LIN {X -0.024,Y -228.688,Z 374.177,A 0.000,B 0.000,C 90.000,E1 31.848} C_DIS
LIN {X 0.017,Y -219.940,Z 374.156,A 0.000,B 0.000,C 90.000,E1 28.025} C_DIS
LIN {X -0.020,Y -212.162,Z 374.134,A 0.000,B 0.000,C 90.000,E1 24.155} C_DIS
LIN {X 0.098,Y -206.724,Z 374.117,A 0.000,B 0.000,C 90.000,E1 20.972} C_DIS
LIN {X -0.105,Y -200.813,Z 374.095,A 0.000,B 0.000,C 90.000,E1 17.040} C_DIS
LIN {X 0.032,Y -196.763,Z 374.077,A 0.000,B 0.000,C 90.000,E1 13.772} C_DIS
LIN {X -0.062,Y -192.666,Z 374.054,A 0.000,B 0.000,C 90.000,E1 9.726} C_DIS
LIN {X -0.090,Y -189.777,Z 374.031,A 0.000,B 0.000,C 90.000,E1 5.625} C_DIS
LIN {X 0.062,Y -187.714,Z 373.993,A 0.000,B 0.000,C 90.000,E1 358.682} C_DIS
LIN {X 0.002,Y -189.474,Z 373.942,A 0.000,B 0.000,C 90.000,E1 349.577} C_DIS
LIN {X -0.013,Y -192.481,Z 373.915,A 0.000,B 0.000,C 90.000,E1 344.629} C_DIS
LIN {X -0.083,Y -196.181,Z 373.892,A 0.000,B 0.000,C 90.000,E1 340.550} C_DIS
LIN {X -0.079,Y -200.966,Z 373.869,A 0.000,B 0.000,C 90.000,E1 336.485} C_DIS
LIN {X -0.043,Y -205.596,Z 373.851,A 0.000,B 0.000,C 90.000,E1 333.256} C_DIS
LIN {X -0.055,Y -212.277,Z 373.829,A 0.000,B 0.000,C 90.000,E1 329.282} C_DIS
LIN {X 0.024,Y -219.465,Z 373.807,A 0.000,B 0.000,C 90.000,E1 325.341} C_DIS
LIN {X -0.061,Y -225.849,Z 373.790,A 0.000,B 0.000,C 90.000,E1 322.271} C_DIS
LIN {X 0.005,Y -234.579,Z 373.769,A 0.000,B 0.000,C 90.000,E1 318.447} C_DIS
LIN {X 0.024,Y -243.663,Z 373.750,A 0.000,B 0.000,C 90.000,E1 315.081} C_DIS
LIN {X -0.040,Y -252.669,Z 373.734,A 0.000,B 0.000,C 90.000,E1 312.162} C_DIS
LIN {X -0.020,Y -262.716,Z 373.718,A 0.000,B 0.000,C 90.000,E1 309.277} C_DIS
LIN {X 0.045,Y -274.656,Z 373.701,A 0.000,B 0.000,C 90.000,E1 306.091} C_DIS
LIN {X -0.160,Y -285.719,Z 373.685,A 0.000,B 0.000,C 90.000,E1 303.372} C_DIS
LIN {X -0.156,Y -299.626,Z 373.668,A 0.000,B 0.000,C 90.000,E1 300.335} C_DIS
LIN {X 0.072,Y -315.196,Z 373.652,A 0.000,B 0.000,C 90.000,E1 297.334} C_DIS
LIN {X 0.056,Y -326.808,Z 373.641,A 0.000,B 0.000,C 90.000,E1 295.412} C_DIS
LIN {X 0.118,Y -339.498,Z 373.631,A 0.000,B 0.000,C 90.000,E1 293.515} C_DIS
LIN {X -0.141,Y -355.051,Z 373.619,A 0.000,B 0.000,C 90.000,E1 291.408} C_DIS
LIN {X 0.226,Y -373.453,Z 373.606,A 0.000,B 0.000,C 90.000,E1 288.960} C_DIS
LIN {X 0.071,Y -398.842,Z 373.590,A 0.000,B 0.000,C 90.000,E1 286.150} C_DIS
LIN {X -0.135,Y -416.958,Z 373.579,A 0.000,B 0.000,C 90.000,E1 284.300} C_DIS
LIN {X -0.034,Y -427.204,Z 373.574,A 0.000,B 0.000,C 90.000,E1 283.244} C_DIS
LIN {X 0.012,Y -437.142,Z 373.568,A 0.000,B 0.000,C 90.000,E1 282.187} C_DIS
LIN {X -0.235,Y -444.156,Z 373.563,A 0.000,B 0.000,C 90.000,E1 281.422} C_DIS
LIN {X -0.195,Y -452.664,Z 373.557,A 0.000,B 0.000,C 90.000,E1 280.366} C_DIS
LIN {X -0.136,Y -460.420,Z 373.552,A 0.000,B 0.000,C 90.000,E1 279.321} C_DIS
LIN {X 0.014,Y -467.426,Z 373.546,A 0.000,B 0.000,C 90.000,E1 278.276} C_DIS
LIN {X 0.186,Y -473.852,Z 373.540,A 0.000,B 0.000,C 90.000,E1 277.239} C_DIS
LIN {X -0.034,Y -479.682,Z 373.535,A 0.000,B 0.000,C 90.000,E1 276.258} C_DIS
LIN {X -0.063,Y -483.421,Z 373.531,A 0.000,B 0.000,C 90.000,E1 275.511} C_DIS
LIN {X 0.114,Y -485.523,Z 373.528,A 0.000,B 0.000,C 90.000,E1 274.992} C_DIS
LIN {X -0.181,Y -487.261,Z 373.525,A 0.000,B 0.000,C 90.000,E1 274.531} C_DIS
LIN {X 0.011,Y -488.621,Z 373.522,A 0.000,B 0.000,C 90.000,E1 274.012} C_DIS
LIN {X 0.181,Y -489.646,Z 373.520,A 0.000,B 0.000,C 90.000,E1 273.498} C_DIS
LIN {X -0.100,Y -490.325,Z 373.517,A 0.000,B 0.000,C 90.000,E1 273.037} C_DIS
LIN {X 0.089,Y -490.720,Z 373.514,A 0.000,B 0.000,C 90.000,E1 272.522} C_DIS
LIN {X -0.206,Y -490.827,Z 373.511,A 0.000,B 0.000,C 90.000,E1 272.064} C_DIS
LIN {X 0.007,Y -490.615,Z 373.509,A 0.000,B 0.000,C 90.000,E1 271.547} C_DIS
LIN {X 0.205,Y -490.110,Z 373.506,A 0.000,B 0.000,C 90.000,E1 271.031} C_DIS
LIN {X -0.086,Y -489.189,Z 373.503,A 0.000,B 0.000,C 90.000,E1 270.573} C_DIS
LIN {X 0.110,Y -487.799,Z 373.500,A 0.000,B 0.000,C 90.000,E1 270.057} C_DIS
LIN {X -0.186,Y -485.830,Z 373.498,A 0.000,B 0.000,C 90.000,E1 269.599} C_DIS
LIN {X 0.148,Y -484.659,Z 373.496,A 0.000,B 0.000,C 90.000,E1 269.312} C_DIS
LIN {X -0.165,Y -481.666,Z 373.494,A 0.000,B 0.000,C 90.000,E1 268.854} C_DIS
LIN {X -0.013,Y -477.763,Z 373.491,A 0.000,B 0.000,C 90.000,E1 268.339} C_DIS
LIN {X -0.165,Y -475.427,Z 373.489,A 0.000,B 0.000,C 90.000,E1 268.108} C_DIS
LIN {X -0.044,Y -469.718,Z 373.487,A 0.000,B 0.000,C 90.000,E1 267.593} C_DIS
LIN {X 0.107,Y -463.235,Z 373.484,A 0.000,B 0.000,C 90.000,E1 267.135} C_DIS
LIN {X 0.020,Y -459.955,Z 373.483,A 0.000,B 0.000,C 90.000,E1 266.963} C_DIS
LIN {X 0.177,Y -452.875,Z 373.481,A 0.000,B 0.000,C 90.000,E1 266.617} C_DIS
LIN {X -0.068,Y -445.562,Z 373.480,A 0.000,B 0.000,C 90.000,E1 266.388} C_DIS
LIN {X 0.108,Y -437.885,Z 373.479,A 0.000,B 0.000,C 90.000,E1 266.159} C_DIS
LIN {X -0.210,Y -429.466,Z 373.478,A 0.000,B 0.000,C 90.000,E1 266.045} C_DIS
LIN {X -0.134,Y -418.655,Z 373.477,A 0.000,B 0.000,C 90.000,E1 265.927} C_DIS
LIN {X 0.128,Y -414.372,Z 373.477,A 0.000,B 0.000,C 90.000,E1 265.869} C_DIS
LIN {X 0.023,Y -180.915,Z 373.477,A 0.000,B 0.000,C 90.000,E1 265.869} C_DIS
LIN {X 0.051,Y -180.822,Z 373.471,A 0.000,B 0.000,C 90.000,E1 264.837} C_DIS
LIN {X -0.054,Y -178.854,Z 373.442,A 0.000,B 0.000,C 90.000,E1 259.634} C_DIS
LIN {X 0.017,Y -175.897,Z 373.414,A 0.000,B 0.000,C 90.000,E1 254.519} C_DIS
LIN {X -0.044,Y -174.574,Z 373.405,A 0.000,B 0.000,C 90.000,E1 252.834} C_DIS
LIN {X -0.008,Y -171.557,Z 373.381,A 0.000,B 0.000,C 90.000,E1 248.539} C_DIS
LIN {X 0.048,Y -167.781,Z 373.357,A 0.000,B 0.000,C 90.000,E1 244.204} C_DIS
LIN {X -0.011,Y -166.494,Z 373.347,A 0.000,B 0.000,C 90.000,E1 242.487} C_DIS
LIN {X -0.015,Y -163.204,Z 373.328,A 0.000,B 0.000,C 90.000,E1 238.997} C_DIS
LIN {X 0.039,Y -161.168,Z 373.313,A 0.000,B 0.000,C 90.000,E1 236.342} C_DIS
LIN {X 0.074,Y -157.183,Z 373.289,A 0.000,B 0.000,C 90.000,E1 231.904} C_DIS
LIN {X -0.003,Y -155.912,Z 373.279,A 0.000,B 0.000,C 90.000,E1 230.150} C_DIS
LIN {X 0.053,Y -152.163,Z 373.254,A 0.000,B 0.000,C 90.000,E1 225.648} C_DIS
LIN {X 0.073,Y -150.412,Z 373.239,A 0.000,B 0.000,C 90.000,E1 222.933} C_DIS
LIN {X 0.004,Y -147.141,Z 373.213,A 0.000,B 0.000,C 90.000,E1 218.418} C_DIS
LIN {X 0.002,Y -145.700,Z 373.198,A 0.000,B 0.000,C 90.000,E1 215.678} C_DIS
LIN {X 0.009,Y -143.083,Z 373.173,A 0.000,B 0.000,C 90.000,E1 211.082} C_DIS
LIN {X 0.014,Y -141.701,Z 373.152,A 0.000,B 0.000,C 90.000,E1 207.385} C_DIS
LIN {X -0.063,Y -139.467,Z 373.116,A 0.000,B 0.000,C 90.000,E1 200.918} C_DIS
LIN {X -0.010,Y -139.200,Z 373.106,A 0.000,B 0.000,C 90.000,E1 199.033} C_DIS
LIN {X 0.054,Y -138.327,Z 373.054,A 0.000,B 0.000,C 90.000,E1 189.670} C_DIS
LIN {X 0.059,Y -139.445,Z 373.007,A 0.000,B 0.000,C 90.000,E1 181.260} C_DIS
LIN {X 0.000,Y -140.983,Z 372.976,A 0.000,B 0.000,C 90.000,E1 175.698} C_DIS
LIN {X -0.051,Y -142.739,Z 372.955,A 0.000,B 0.000,C 90.000,E1 172.008} C_DIS
LIN {X 0.047,Y -145.131,Z 372.930,A 0.000,B 0.000,C 90.000,E1 167.353} C_DIS
LIN {X 0.042,Y -147.754,Z 372.909,A 0.000,B 0.000,C 90.000,E1 163.685} C_DIS
LIN {X -0.020,Y -150.424,Z 372.889,A 0.000,B 0.000,C 90.000,E1 160.061} C_DIS
LIN {X -0.005,Y -153.865,Z 372.869,A 0.000,B 0.000,C 90.000,E1 156.433} C_DIS
LIN {X -0.088,Y -157.276,Z 372.849,A 0.000,B 0.000,C 90.000,E1 152.871} C_DIS
LIN {X -0.011,Y -161.454,Z 372.829,A 0.000,B 0.000,C 90.000,E1 149.282} C_DIS
LIN {X -0.004,Y -165.655,Z 372.810,A 0.000,B 0.000,C 90.000,E1 145.754} C_DIS
LIN {X -0.022,Y -170.590,Z 372.790,A 0.000,B 0.000,C 90.000,E1 142.271} C_DIS
LIN {X 0.017,Y -175.468,Z 372.771,A 0.000,B 0.000,C 90.000,E1 138.809} C_DIS
LIN {X 0.000,Y -181.090,Z 372.752,A 0.000,B 0.000,C 90.000,E1 135.405} C_DIS
LIN {X -0.010,Y -186.531,Z 372.734,A 0.000,B 0.000,C 90.000,E1 132.043} C_DIS
LIN {X -0.069,Y -191.149,Z 372.720,A 0.000,B 0.000,C 90.000,E1 129.564} C_DIS
LIN {X 0.009,Y -196.950,Z 372.701,A 0.000,B 0.000,C 90.000,E1 126.251} C_DIS
LIN {X -0.085,Y -199.016,Z 372.696,A 0.000,B 0.000,C 90.000,E1 125.231} C_DIS
LIN {X 0.067,Y -298.976,Z 372.696,A 0.000,B 0.000,C 90.000,E1 125.185} C_DIS
LIN {X -0.082,Y -300.521,Z 372.695,A 0.000,B 0.000,C 90.000,E1 125.185} C_DIS
LIN {X -0.007,Y -305.764,Z 372.694,A 0.000,B 0.000,C 90.000,E1 124.898} C_DIS
LIN {X 0.070,Y -308.564,Z 372.692,A 0.000,B 0.000,C 90.000,E1 124.612} C_DIS
LIN {X 0.009,Y -312.276,Z 372.689,A 0.000,B 0.000,C 90.000,E1 124.072} C_DIS
LIN {X -0.208,Y -313.814,Z 372.688,A 0.000,B 0.000,C 90.000,E1 123.785} C_DIS
LIN {X 0.077,Y -320.564,Z 372.677,A 0.000,B 0.000,C 90.000,E1 121.799} C_DIS
LIN {X 0.040,Y -331.559,Z 372.661,A 0.000,B 0.000,C 90.000,E1 118.949} C_DIS
LIN {X -0.002,Y -343.956,Z 372.645,A 0.000,B 0.000,C 90.000,E1 116.155} C_DIS
LIN {X 0.123,Y -356.250,Z 372.632,A 0.000,B 0.000,C 90.000,E1 113.695} C_DIS
LIN {X -0.057,Y -369.833,Z 372.618,A 0.000,B 0.000,C 90.000,E1 111.334} C_DIS
LIN {X 0.186,Y -384.804,Z 372.605,A 0.000,B 0.000,C 90.000,E1 108.960} C_DIS
LIN {X 0.205,Y -401.275,Z 372.593,A 0.000,B 0.000,C 90.000,E1 106.677} C_DIS
LIN {X 0.020,Y -419.367,Z 372.580,A 0.000,B 0.000,C 90.000,E1 104.481} C_DIS
LIN {X -0.114,Y -439.036,Z 372.569,A 0.000,B 0.000,C 90.000,E1 102.355} C_DIS
LIN {X -0.027,Y -459.428,Z 372.558,A 0.000,B 0.000,C 90.000,E1 100.366} C_DIS
LIN {X -0.068,Y -482.997,Z 372.546,A 0.000,B 0.000,C 90.000,E1 98.341} C_DIS
LIN {X -0.008,Y -490.879,Z 372.543,A 0.000,B 0.000,C 90.000,E1 97.701} C_DIS
LIN {X 0.157,Y -492.885,Z 372.542,A 0.000,B 0.000,C 90.000,E1 97.473} C_DIS
LIN {X 0.059,Y -494.681,Z 372.540,A 0.000,B 0.000,C 90.000,E1 97.239} C_DIS
LIN {X -0.042,Y -496.029,Z 372.539,A 0.000,B 0.000,C 90.000,E1 97.004} C_DIS
LIN {X 0.210,Y -497.710,Z 372.536,A 0.000,B 0.000,C 90.000,E1 96.486} C_DIS
LIN {X -0.078,Y -498.302,Z 372.533,A 0.000,B 0.000,C 90.000,E1 96.030} C_DIS
LIN {X 0.194,Y -497.899,Z 372.531,A 0.000,B 0.000,C 90.000,E1 95.511} C_DIS
LIN {X -0.027,Y -496.437,Z 372.528,A 0.000,B 0.000,C 90.000,E1 95.049} C_DIS
LIN {X -0.159,Y -495.229,Z 372.527,A 0.000,B 0.000,C 90.000,E1 94.821} C_DIS
LIN {X -0.035,Y -490.066,Z 372.523,A 0.000,B 0.000,C 90.000,E1 94.073} C_DIS
LIN {X -0.087,Y -482.358,Z 372.517,A 0.000,B 0.000,C 90.000,E1 93.094} C_DIS
LIN {X -0.201,Y -460.635,Z 372.502,A 0.000,B 0.000,C 90.000,E1 90.344} C_DIS
LIN {X 0.204,Y -442.378,Z 372.487,A 0.000,B 0.000,C 90.000,E1 87.707} C_DIS
LIN {X 0.098,Y -420.907,Z 372.468,A 0.000,B 0.000,C 90.000,E1 84.261} C_DIS
LIN {X -0.157,Y -407.216,Z 372.455,A 0.000,B 0.000,C 90.000,E1 81.837} C_DIS
LIN {X 0.072,Y -395.395,Z 372.442,A 0.000,B 0.000,C 90.000,E1 79.577} C_DIS
LIN {X 0.110,Y -385.202,Z 372.431,A 0.000,B 0.000,C 90.000,E1 77.589} C_DIS
LIN {X 0.118,Y -372.056,Z 372.417,A 0.000,B 0.000,C 90.000,E1 74.991} C_DIS
LIN {X -0.087,Y -360.570,Z 372.404,A 0.000,B 0.000,C 90.000,E1 72.670} C_DIS
LIN {X 0.067,Y -350.621,Z 372.392,A 0.000,B 0.000,C 90.000,E1 70.550} C_DIS
LIN {X 0.131,Y -338.104,Z 372.377,A 0.000,B 0.000,C 90.000,E1 67.794} C_DIS
LIN {X -0.137,Y -323.705,Z 372.358,A 0.000,B 0.000,C 90.000,E1 64.409} C_DIS
LIN {X 0.065,Y -311.675,Z 372.340,A 0.000,B 0.000,C 90.000,E1 61.179} C_DIS
LIN {X 0.081,Y -300.462,Z 372.322,A 0.000,B 0.000,C 90.000,E1 57.916} C_DIS
LIN {X 0.017,Y -290.095,Z 372.303,A 0.000,B 0.000,C 90.000,E1 54.609} C_DIS
LIN {X 0.042,Y -282.469,Z 372.288,A 0.000,B 0.000,C 90.000,E1 51.904} C_DIS
LIN {X -0.003,Y -275.091,Z 372.273,A 0.000,B 0.000,C 90.000,E1 49.175} C_DIS
LIN {X 0.095,Y -267.499,Z 372.258,A 0.000,B 0.000,C 90.000,E1 46.377} C_DIS
LIN {X -0.002,Y -259.878,Z 372.242,A 0.000,B 0.000,C 90.000,E1 43.581} C_DIS
LIN {X 0.029,Y -254.052,Z 372.230,A 0.000,B 0.000,C 90.000,E1 41.434} C_DIS
LIN {X 0.020,Y -246.068,Z 372.214,A 0.000,B 0.000,C 90.000,E1 38.543} C_DIS
LIN {X 0.051,Y -238.246,Z 372.198,A 0.000,B 0.000,C 90.000,E1 35.598} C_DIS
LIN {X 0.000,Y -230.723,Z 372.181,A 0.000,B 0.000,C 90.000,E1 32.625} C_DIS
LIN {X 0.021,Y -223.507,Z 372.164,A 0.000,B 0.000,C 90.000,E1 29.589} C_DIS
LIN {X 0.111,Y -216.892,Z 372.147,A 0.000,B 0.000,C 90.000,E1 26.488} C_DIS
LIN {X 0.043,Y -210.870,Z 372.130,A 0.000,B 0.000,C 90.000,E1 23.387} C_DIS
LIN {X -0.030,Y -205.581,Z 372.112,A 0.000,B 0.000,C 90.000,E1 20.248} C_DIS
LIN {X -0.069,Y -199.789,Z 372.090,A 0.000,B 0.000,C 90.000,E1 16.260} C_DIS
LIN {X -0.007,Y -195.947,Z 372.072,A 0.000,B 0.000,C 90.000,E1 13.008} C_DIS
LIN {X 0.027,Y -192.016,Z 372.050,A 0.000,B 0.000,C 90.000,E1 8.916} C_DIS
LIN {X 0.091,Y -188.997,Z 372.022,A 0.000,B 0.000,C 90.000,E1 3.955} C_DIS
LIN {X -0.067,Y -188.058,Z 371.965,A 0.000,B 0.000,C 90.000,E1 353.742} C_DIS
LIN {X -0.066,Y -190.713,Z 371.928,A 0.000,B 0.000,C 90.000,E1 347.117} C_DIS
LIN {X -0.070,Y -194.489,Z 371.901,A 0.000,B 0.000,C 90.000,E1 342.181} C_DIS
LIN {X -0.076,Y -198.867,Z 371.878,A 0.000,B 0.000,C 90.000,E1 338.103} C_DIS
LIN {X 0.006,Y -203.091,Z 371.860,A 0.000,B 0.000,C 90.000,E1 334.845} C_DIS
LIN {X 0.007,Y -209.442,Z 371.838,A 0.000,B 0.000,C 90.000,E1 330.845} C_DIS
LIN {X -0.039,Y -216.434,Z 371.816,A 0.000,B 0.000,C 90.000,E1 326.914} C_DIS
LIN {X 0.031,Y -222.445,Z 371.799,A 0.000,B 0.000,C 90.000,E1 323.783} C_DIS
LIN {X -0.015,Y -229.178,Z 371.782,A 0.000,B 0.000,C 90.000,E1 320.723} C_DIS
LIN {X 0.018,Y -237.396,Z 371.763,A 0.000,B 0.000,C 90.000,E1 317.310} C_DIS
LIN {X 0.115,Y -246.852,Z 371.744,A 0.000,B 0.000,C 90.000,E1 313.947} C_DIS
LIN {X 0.111,Y -253.839,Z 371.732,A 0.000,B 0.000,C 90.000,E1 311.757} C_DIS
LIN {X -0.006,Y -263.914,Z 371.716,A 0.000,B 0.000,C 90.000,E1 308.910} C_DIS
LIN {X 0.007,Y -274.572,Z 371.701,A 0.000,B 0.000,C 90.000,E1 306.091} C_DIS
LIN {X 0.194,Y -285.683,Z 371.685,A 0.000,B 0.000,C 90.000,E1 303.293} C_DIS
LIN {X 0.059,Y -299.634,Z 371.668,A 0.000,B 0.000,C 90.000,E1 300.285} C_DIS
LIN {X 0.027,Y -315.307,Z 371.652,A 0.000,B 0.000,C 90.000,E1 297.334} C_DIS
LIN {X 0.074,Y -324.949,Z 371.643,A 0.000,B 0.000,C 90.000,E1 295.720} C_DIS
LIN {X 0.076,Y -339.679,Z 371.631,A 0.000,B 0.000,C 90.000,E1 293.515} C_DIS
LIN {X -0.181,Y -355.254,Z 371.619,A 0.000,B 0.000,C 90.000,E1 291.408} C_DIS
LIN {X 0.098,Y -371.302,Z 371.607,A 0.000,B 0.000,C 90.000,E1 289.268} C_DIS
LIN {X -0.168,Y -386.166,Z 371.598,A 0.000,B 0.000,C 90.000,E1 287.583} C_DIS
LIN {X 0.020,Y -404.328,Z 371.587,A 0.000,B 0.000,C 90.000,E1 285.607} C_DIS
LIN {X -0.243,Y -422.490,Z 371.576,A 0.000,B 0.000,C 90.000,E1 283.772} C_DIS
LIN {X 0.041,Y -432.438,Z 371.571,A 0.000,B 0.000,C 90.000,E1 282.703} C_DIS
LIN {X -0.206,Y -439.634,Z 371.566,A 0.000,B 0.000,C 90.000,E1 281.951} C_DIS
LIN {X 0.063,Y -446.350,Z 371.562,A 0.000,B 0.000,C 90.000,E1 281.130} C_DIS
LIN {X 0.134,Y -454.649,Z 371.556,A 0.000,B 0.000,C 90.000,E1 280.074} C_DIS
LIN {X 0.221,Y -462.124,Z 371.550,A 0.000,B 0.000,C 90.000,E1 279.029} C_DIS
LIN {X -0.134,Y -469.004,Z 371.545,A 0.000,B 0.000,C 90.000,E1 278.049} C_DIS
LIN {X 0.119,Y -475.230,Z 371.539,A 0.000,B 0.000,C 90.000,E1 277.004} C_DIS
LIN {X 0.051,Y -479.565,Z 371.535,A 0.000,B 0.000,C 90.000,E1 276.258} C_DIS
LIN {X 0.020,Y -483.335,Z 371.531,A 0.000,B 0.000,C 90.000,E1 275.511} C_DIS
LIN {X 0.198,Y -485.450,Z 371.528,A 0.000,B 0.000,C 90.000,E1 274.992} C_DIS
LIN {X -0.098,Y -487.170,Z 371.525,A 0.000,B 0.000,C 90.000,E1 274.531} C_DIS
LIN {X 0.094,Y -488.544,Z 371.522,A 0.000,B 0.000,C 90.000,E1 274.012} C_DIS
LIN {X -0.225,Y -489.539,Z 371.520,A 0.000,B 0.000,C 90.000,E1 273.555} C_DIS
LIN {X -0.018,Y -490.211,Z 371.517,A 0.000,B 0.000,C 90.000,E1 273.037} C_DIS
LIN {X 0.171,Y -490.608,Z 371.514,A 0.000,B 0.000,C 90.000,E1 272.522} C_DIS
LIN {X -0.125,Y -490.705,Z 371.511,A 0.000,B 0.000,C 90.000,E1 272.064} C_DIS
LIN {X 0.088,Y -490.499,Z 371.509,A 0.000,B 0.000,C 90.000,E1 271.547} C_DIS
LIN {X -0.204,Y -489.981,Z 371.506,A 0.000,B 0.000,C 90.000,E1 271.088} C_DIS
LIN {X -0.006,Y -489.061,Z 371.503,A 0.000,B 0.000,C 90.000,E1 270.573} C_DIS
LIN {X 0.188,Y -487.719,Z 371.500,A 0.000,B 0.000,C 90.000,E1 270.057} C_DIS
LIN {X -0.109,Y -485.816,Z 371.498,A 0.000,B 0.000,C 90.000,E1 269.599} C_DIS
LIN {X 0.072,Y -483.222,Z 371.495,A 0.000,B 0.000,C 90.000,E1 269.083} C_DIS
LIN {X -0.089,Y -481.681,Z 371.494,A 0.000,B 0.000,C 90.000,E1 268.854} C_DIS
LIN {X 0.062,Y -477.860,Z 371.491,A 0.000,B 0.000,C 90.000,E1 268.339} C_DIS
LIN {X -0.090,Y -475.546,Z 371.489,A 0.000,B 0.000,C 90.000,E1 268.108} C_DIS
LIN {X 0.208,Y -472.879,Z 371.488,A 0.000,B 0.000,C 90.000,E1 267.822} C_DIS
LIN {X 0.098,Y -466.953,Z 371.485,A 0.000,B 0.000,C 90.000,E1 267.364} C_DIS
LIN {X 0.107,Y -460.313,Z 371.483,A 0.000,B 0.000,C 90.000,E1 266.963} C_DIS
LIN {X -0.206,Y -453.387,Z 371.481,A 0.000,B 0.000,C 90.000,E1 266.674} C_DIS
LIN {X -0.054,Y -445.982,Z 371.480,A 0.000,B 0.000,C 90.000,E1 266.388} C_DIS
LIN {X 0.104,Y -438.346,Z 371.479,A 0.000,B 0.000,C 90.000,E1 266.159} C_DIS
LIN {X -0.225,Y -429.948,Z 371.478,A 0.000,B 0.000,C 90.000,E1 266.045} C_DIS
LIN {X -0.156,Y -419.101,Z 371.477,A 0.000,B 0.000,C 90.000,E1 265.927} C_DIS
LIN {X 0.106,Y -415.628,Z 371.477,A 0.000,B 0.000,C 90.000,E1 265.869} C_DIS
LIN {X 0.012,Y -180.915,Z 371.477,A 0.000,B 0.000,C 90.000,E1 265.869} C_DIS
LIN {X 0.040,Y -180.821,Z 371.471,A 0.000,B 0.000,C 90.000,E1 264.837} C_DIS
LIN {X -0.065,Y -178.852,Z 371.442,A 0.000,B 0.000,C 90.000,E1 259.634} C_DIS
LIN {X 0.007,Y -175.896,Z 371.414,A 0.000,B 0.000,C 90.000,E1 254.519} C_DIS
LIN {X -0.055,Y -174.571,Z 371.405,A 0.000,B 0.000,C 90.000,E1 252.834} C_DIS
LIN {X -0.019,Y -171.554,Z 371.381,A 0.000,B 0.000,C 90.000,E1 248.539} C_DIS
LIN {X 0.037,Y -167.778,Z 371.357,A 0.000,B 0.000,C 90.000,E1 244.204} C_DIS
LIN {X -0.021,Y -166.490,Z 371.347,A 0.000,B 0.000,C 90.000,E1 242.487} C_DIS
LIN {X -0.026,Y -163.200,Z 371.328,A 0.000,B 0.000,C 90.000,E1 238.997} C_DIS
LIN {X 0.028,Y -161.164,Z 371.313,A 0.000,B 0.000,C 90.000,E1 236.342} C_DIS
LIN {X 0.064,Y -157.180,Z 371.288,A 0.000,B 0.000,C 90.000,E1 231.904} C_DIS
LIN {X -0.014,Y -155.910,Z 371.279,A 0.000,B 0.000,C 90.000,E1 230.150} C_DIS
LIN {X 0.043,Y -152.161,Z 371.254,A 0.000,B 0.000,C 90.000,E1 225.648} C_DIS
LIN {X 0.063,Y -150.410,Z 371.239,A 0.000,B 0.000,C 90.000,E1 222.933} C_DIS
LIN {X 0.086,Y -147.139,Z 371.213,A 0.000,B 0.000,C 90.000,E1 218.382} C_DIS
LIN {X -0.008,Y -145.698,Z 371.198,A 0.000,B 0.000,C 90.000,E1 215.678} C_DIS
LIN {X 0.000,Y -143.082,Z 371.173,A 0.000,B 0.000,C 90.000,E1 211.082} C_DIS
LIN {X 0.004,Y -141.699,Z 371.152,A 0.000,B 0.000,C 90.000,E1 207.385} C_DIS
LIN {X -0.073,Y -139.466,Z 371.116,A 0.000,B 0.000,C 90.000,E1 200.918} C_DIS
LIN {X -0.019,Y -139.199,Z 371.106,A 0.000,B 0.000,C 90.000,E1 199.033} C_DIS
LIN {X 0.045,Y -138.327,Z 371.054,A 0.000,B 0.000,C 90.000,E1 189.670} C_DIS
LIN {X 0.050,Y -139.446,Z 371.007,A 0.000,B 0.000,C 90.000,E1 181.260} C_DIS
LIN {X -0.010,Y -140.985,Z 370.976,A 0.000,B 0.000,C 90.000,E1 175.698} C_DIS
LIN {X -0.060,Y -142.740,Z 370.955,A 0.000,B 0.000,C 90.000,E1 172.008} C_DIS
LIN {X 0.038,Y -145.133,Z 370.930,A 0.000,B 0.000,C 90.000,E1 167.353} C_DIS
LIN {X 0.031,Y -147.756,Z 370.909,A 0.000,B 0.000,C 90.000,E1 163.685} C_DIS
LIN {X -0.029,Y -150.426,Z 370.889,A 0.000,B 0.000,C 90.000,E1 160.061} C_DIS
LIN {X -0.015,Y -153.869,Z 370.869,A 0.000,B 0.000,C 90.000,E1 156.433} C_DIS
LIN {X 0.042,Y -157.280,Z 370.849,A 0.000,B 0.000,C 90.000,E1 152.820} C_DIS
LIN {X -0.021,Y -161.459,Z 370.829,A 0.000,B 0.000,C 90.000,E1 149.282} C_DIS
LIN {X -0.015,Y -165.660,Z 370.810,A 0.000,B 0.000,C 90.000,E1 145.754} C_DIS
LIN {X -0.033,Y -170.596,Z 370.790,A 0.000,B 0.000,C 90.000,E1 142.271} C_DIS
LIN {X 0.005,Y -175.472,Z 370.771,A 0.000,B 0.000,C 90.000,E1 138.809} C_DIS
LIN {X -0.011,Y -181.095,Z 370.752,A 0.000,B 0.000,C 90.000,E1 135.405} C_DIS
LIN {X -0.022,Y -186.538,Z 370.734,A 0.000,B 0.000,C 90.000,E1 132.043} C_DIS
LIN {X -0.081,Y -191.154,Z 370.720,A 0.000,B 0.000,C 90.000,E1 129.564} C_DIS
LIN {X -0.003,Y -196.957,Z 370.701,A 0.000,B 0.000,C 90.000,E1 126.251} C_DIS
LIN {X 0.000,Y -199.129,Z 370.695,A 0.000,B 0.000,C 90.000,E1 125.152} C_DIS
LIN {X -0.036,Y -298.758,Z 370.695,A 0.000,B 0.000,C 90.000,E1 125.152} C_DIS
LIN {X -0.018,Y -301.092,Z 370.695,A 0.000,B 0.000,C 90.000,E1 125.105} C_DIS
LIN {X -0.022,Y -305.657,Z 370.694,A 0.000,B 0.000,C 90.000,E1 124.865} C_DIS
LIN {X 0.052,Y -308.254,Z 370.692,A 0.000,B 0.000,C 90.000,E1 124.612} C_DIS
LIN {X -0.151,Y -312.031,Z 370.689,A 0.000,B 0.000,C 90.000,E1 124.119} C_DIS
LIN {X -0.109,Y -313.659,Z 370.688,A 0.000,B 0.000,C 90.000,E1 123.785} C_DIS
LIN {X 0.166,Y -316.023,Z 370.684,A 0.000,B 0.000,C 90.000,E1 123.086} C_DIS
LIN {X -0.116,Y -326.417,Z 370.668,A 0.000,B 0.000,C 90.000,E1 120.256} C_DIS
LIN {X 0.146,Y -338.167,Z 370.652,A 0.000,B 0.000,C 90.000,E1 117.385} C_DIS
LIN {X -0.018,Y -351.389,Z 370.637,A 0.000,B 0.000,C 90.000,E1 114.643} C_DIS
LIN {X 0.159,Y -364.468,Z 370.624,A 0.000,B 0.000,C 90.000,E1 112.206} C_DIS
LIN {X -0.080,Y -378.897,Z 370.610,A 0.000,B 0.000,C 90.000,E1 109.885} C_DIS
LIN {X -0.089,Y -394.782,Z 370.598,A 0.000,B 0.000,C 90.000,E1 107.583} C_DIS
LIN {X 0.065,Y -412.240,Z 370.585,A 0.000,B 0.000,C 90.000,E1 105.315} C_DIS
LIN {X 0.155,Y -431.393,Z 370.573,A 0.000,B 0.000,C 90.000,E1 103.119} C_DIS
LIN {X 0.169,Y -451.570,Z 370.562,A 0.000,B 0.000,C 90.000,E1 101.074} C_DIS
LIN {X 0.114,Y -472.289,Z 370.551,A 0.000,B 0.000,C 90.000,E1 99.208} C_DIS
LIN {X 0.082,Y -490.755,Z 370.543,A 0.000,B 0.000,C 90.000,E1 97.701} C_DIS
LIN {X -0.243,Y -492.842,Z 370.542,A 0.000,B 0.000,C 90.000,E1 97.530} C_DIS
LIN {X 0.180,Y -494.676,Z 370.540,A 0.000,B 0.000,C 90.000,E1 97.239} C_DIS
LIN {X 0.113,Y -496.060,Z 370.539,A 0.000,B 0.000,C 90.000,E1 97.004} C_DIS
LIN {X -0.130,Y -497.831,Z 370.536,A 0.000,B 0.000,C 90.000,E1 96.543} C_DIS
LIN {X 0.077,Y -498.496,Z 370.534,A 0.000,B 0.000,C 90.000,E1 96.030} C_DIS
LIN {X -0.146,Y -498.165,Z 370.531,A 0.000,B 0.000,C 90.000,E1 95.568} C_DIS
LIN {X 0.129,Y -496.785,Z 370.528,A 0.000,B 0.000,C 90.000,E1 95.049} C_DIS
LIN {X -0.003,Y -495.629,Z 370.527,A 0.000,B 0.000,C 90.000,E1 94.821} C_DIS
LIN {X -0.232,Y -492.321,Z 370.524,A 0.000,B 0.000,C 90.000,E1 94.359} C_DIS
LIN {X 0.199,Y -484.814,Z 370.519,A 0.000,B 0.000,C 90.000,E1 93.326} C_DIS
LIN {X 0.184,Y -472.799,Z 370.510,A 0.000,B 0.000,C 90.000,E1 91.835} C_DIS
LIN {X 0.004,Y -449.877,Z 370.493,A 0.000,B 0.000,C 90.000,E1 88.797} C_DIS
LIN {X 0.141,Y -427.642,Z 370.474,A 0.000,B 0.000,C 90.000,E1 85.355} C_DIS
LIN {X -0.086,Y -409.071,Z 370.456,A 0.000,B 0.000,C 90.000,E1 82.129} C_DIS
LIN {X -0.131,Y -395.773,Z 370.442,A 0.000,B 0.000,C 90.000,E1 79.634} C_DIS
LIN {X -0.037,Y -384.102,Z 370.430,A 0.000,B 0.000,C 90.000,E1 77.353} C_DIS
LIN {X -0.049,Y -372.424,Z 370.417,A 0.000,B 0.000,C 90.000,E1 75.046} C_DIS
LIN {X 0.109,Y -360.933,Z 370.404,A 0.000,B 0.000,C 90.000,E1 72.670} C_DIS
LIN {X -0.066,Y -350.960,Z 370.392,A 0.000,B 0.000,C 90.000,E1 70.604} C_DIS
LIN {X 0.016,Y -338.382,Z 370.377,A 0.000,B 0.000,C 90.000,E1 67.847} C_DIS
LIN {X 0.063,Y -323.950,Z 370.358,A 0.000,B 0.000,C 90.000,E1 64.409} C_DIS
LIN {X -0.074,Y -313.094,Z 370.342,A 0.000,B 0.000,C 90.000,E1 61.563} C_DIS
LIN {X -0.134,Y -300.706,Z 370.322,A 0.000,B 0.000,C 90.000,E1 57.995} C_DIS
LIN {X 0.044,Y -290.326,Z 370.304,A 0.000,B 0.000,C 90.000,E1 54.642} C_DIS
LIN {X 0.014,Y -282.689,Z 370.289,A 0.000,B 0.000,C 90.000,E1 51.949} C_DIS
LIN {X -0.027,Y -277.135,Z 370.277,A 0.000,B 0.000,C 90.000,E1 49.908} C_DIS
LIN {X -0.029,Y -271.493,Z 370.266,A 0.000,B 0.000,C 90.000,E1 47.838} C_DIS
LIN {X 0.046,Y -265.811,Z 370.254,A 0.000,B 0.000,C 90.000,E1 45.729} C_DIS
LIN {X -0.090,Y -258.174,Z 370.238,A 0.000,B 0.000,C 90.000,E1 42.933} C_DIS
LIN {X -0.071,Y -252.294,Z 370.226,A 0.000,B 0.000,C 90.000,E1 40.782} C_DIS
LIN {X -0.114,Y -244.356,Z 370.210,A 0.000,B 0.000,C 90.000,E1 37.890} C_DIS
LIN {X 0.070,Y -236.592,Z 370.194,A 0.000,B 0.000,C 90.000,E1 34.898} C_DIS
LIN {X -0.024,Y -229.103,Z 370.177,A 0.000,B 0.000,C 90.000,E1 31.926} C_DIS
LIN {X 0.031,Y -221.996,Z 370.160,A 0.000,B 0.000,C 90.000,E1 28.871} C_DIS
LIN {X -0.047,Y -213.969,Z 370.139,A 0.000,B 0.000,C 90.000,E1 25.027} C_DIS
LIN {X -0.076,Y -208.297,Z 370.122,A 0.000,B 0.000,C 90.000,E1 21.897} C_DIS
LIN {X -0.089,Y -203.318,Z 370.104,A 0.000,B 0.000,C 90.000,E1 18.725} C_DIS
LIN {X 0.028,Y -198.843,Z 370.086,A 0.000,B 0.000,C 90.000,E1 15.481} C_DIS
LIN {X 0.036,Y -194.348,Z 370.064,A 0.000,B 0.000,C 90.000,E1 11.422} C_DIS
LIN {X -0.049,Y -190.846,Z 370.041,A 0.000,B 0.000,C 90.000,E1 7.352} C_DIS
LIN {X 0.035,Y -188.140,Z 370.009,A 0.000,B 0.000,C 90.000,E1 1.547} C_DIS
LIN {X 0.032,Y -189.398,Z 369.942,A 0.000,B 0.000,C 90.000,E1 349.567} C_DIS
LIN {X -0.021,Y -192.341,Z 369.915,A 0.000,B 0.000,C 90.000,E1 344.629} C_DIS
LIN {X -0.095,Y -196.034,Z 369.892,A 0.000,B 0.000,C 90.000,E1 340.550} C_DIS
LIN {X -0.097,Y -200.811,Z 369.869,A 0.000,B 0.000,C 90.000,E1 336.485} C_DIS
LIN {X -0.065,Y -205.431,Z 369.851,A 0.000,B 0.000,C 90.000,E1 333.256} C_DIS
LIN {X 0.024,Y -212.092,Z 369.829,A 0.000,B 0.000,C 90.000,E1 329.253} C_DIS
LIN {X -0.011,Y -219.262,Z 369.807,A 0.000,B 0.000,C 90.000,E1 325.341} C_DIS
LIN {X -0.102,Y -225.682,Z 369.790,A 0.000,B 0.000,C 90.000,E1 322.271} C_DIS
LIN {X -0.043,Y -234.424,Z 369.769,A 0.000,B 0.000,C 90.000,E1 318.447} C_DIS
LIN {X -0.031,Y -243.523,Z 369.750,A 0.000,B 0.000,C 90.000,E1 315.081} C_DIS
LIN {X 0.070,Y -252.537,Z 369.734,A 0.000,B 0.000,C 90.000,E1 312.123} C_DIS
LIN {X -0.086,Y -262.544,Z 369.718,A 0.000,B 0.000,C 90.000,E1 309.277} C_DIS
LIN {X -0.029,Y -274.491,Z 369.700,A 0.000,B 0.000,C 90.000,E1 306.091} C_DIS
LIN {X 0.040,Y -284.184,Z 369.687,A 0.000,B 0.000,C 90.000,E1 303.658} C_DIS
LIN {X 0.018,Y -299.654,Z 369.668,A 0.000,B 0.000,C 90.000,E1 300.285} C_DIS
LIN {X 0.083,Y -313.592,Z 369.654,A 0.000,B 0.000,C 90.000,E1 297.641} C_DIS
LIN {X -0.048,Y -323.116,Z 369.645,A 0.000,B 0.000,C 90.000,E1 296.052} C_DIS
LIN {X 0.057,Y -337.672,Z 369.632,A 0.000,B 0.000,C 90.000,E1 293.823} C_DIS
LIN {X 0.077,Y -353.244,Z 369.620,A 0.000,B 0.000,C 90.000,E1 291.663} C_DIS
LIN {X 0.064,Y -371.557,Z 369.607,A 0.000,B 0.000,C 90.000,E1 289.268} C_DIS
LIN {X 0.041,Y -388.930,Z 369.596,A 0.000,B 0.000,C 90.000,E1 287.275} C_DIS
LIN {X -0.084,Y -406.919,Z 369.585,A 0.000,B 0.000,C 90.000,E1 285.371} C_DIS
LIN {X -0.062,Y -422.426,Z 369.576,A 0.000,B 0.000,C 90.000,E1 283.772} C_DIS
LIN {X -0.209,Y -430.022,Z 369.572,A 0.000,B 0.000,C 90.000,E1 283.008} C_DIS
LIN {X 0.014,Y -437.375,Z 369.568,A 0.000,B 0.000,C 90.000,E1 282.187} C_DIS
LIN {X -0.232,Y -444.322,Z 369.563,A 0.000,B 0.000,C 90.000,E1 281.422} C_DIS
LIN {X -0.189,Y -452.716,Z 369.557,A 0.000,B 0.000,C 90.000,E1 280.366} C_DIS
LIN {X 0.051,Y -458.528,Z 369.553,A 0.000,B 0.000,C 90.000,E1 279.557} C_DIS
LIN {X 0.186,Y -465.681,Z 369.547,A 0.000,B 0.000,C 90.000,E1 278.511} C_DIS
LIN {X -0.126,Y -472.185,Z 369.542,A 0.000,B 0.000,C 90.000,E1 277.530} C_DIS
LIN {X 0.164,Y -478.144,Z 369.536,A 0.000,B 0.000,C 90.000,E1 276.486} C_DIS
LIN {X 0.124,Y -482.137,Z 369.532,A 0.000,B 0.000,C 90.000,E1 275.739} C_DIS
LIN {X -0.191,Y -484.418,Z 369.529,A 0.000,B 0.000,C 90.000,E1 275.277} C_DIS
LIN {X -0.179,Y -487.133,Z 369.525,A 0.000,B 0.000,C 90.000,E1 274.531} C_DIS
LIN {X 0.012,Y -488.472,Z 369.522,A 0.000,B 0.000,C 90.000,E1 274.012} C_DIS
LIN {X 0.182,Y -489.462,Z 369.520,A 0.000,B 0.000,C 90.000,E1 273.498} C_DIS
LIN {X -0.099,Y -490.090,Z 369.517,A 0.000,B 0.000,C 90.000,E1 273.037} C_DIS
LIN {X 0.088,Y -490.468,Z 369.514,A 0.000,B 0.000,C 90.000,E1 272.522} C_DIS
LIN {X -0.208,Y -490.560,Z 369.511,A 0.000,B 0.000,C 90.000,E1 272.064} C_DIS
LIN {X 0.003,Y -490.349,Z 369.509,A 0.000,B 0.000,C 90.000,E1 271.547} C_DIS
LIN {X 0.200,Y -489.798,Z 369.506,A 0.000,B 0.000,C 90.000,E1 271.031} C_DIS
LIN {X -0.093,Y -488.890,Z 369.503,A 0.000,B 0.000,C 90.000,E1 270.573} C_DIS
LIN {X 0.101,Y -487.539,Z 369.500,A 0.000,B 0.000,C 90.000,E1 270.057} C_DIS
LIN {X -0.196,Y -485.624,Z 369.498,A 0.000,B 0.000,C 90.000,E1 269.599} C_DIS
LIN {X -0.016,Y -483.072,Z 369.495,A 0.000,B 0.000,C 90.000,E1 269.083} C_DIS
LIN {X 0.143,Y -479.768,Z 369.492,A 0.000,B 0.000,C 90.000,E1 268.568} C_DIS
LIN {X -0.026,Y -477.751,Z 369.491,A 0.000,B 0.000,C 90.000,E1 268.339} C_DIS
LIN {X -0.178,Y -475.453,Z 369.489,A 0.000,B 0.000,C 90.000,E1 268.108} C_DIS
LIN {X -0.057,Y -469.868,Z 369.487,A 0.000,B 0.000,C 90.000,E1 267.593} C_DIS
LIN {X 0.014,Y -463.325,Z 369.484,A 0.000,B 0.000,C 90.000,E1 267.135} C_DIS
LIN {X -0.154,Y -456.402,Z 369.482,A 0.000,B 0.000,C 90.000,E1 266.788} C_DIS
LIN {X 0.194,Y -448.969,Z 369.480,A 0.000,B 0.000,C 90.000,E1 266.445} C_DIS
LIN {X 0.171,Y -441.525,Z 369.479,A 0.000,B 0.000,C 90.000,E1 266.216} C_DIS
LIN {X 0.098,Y -433.241,Z 369.478,A 0.000,B 0.000,C 90.000,E1 266.045} C_DIS
LIN {X 0.035,Y -423.586,Z 369.477,A 0.000,B 0.000,C 90.000,E1 265.927} C_DIS
LIN {X 0.000,Y -412.395,Z 369.477,A 0.000,B 0.000,C 90.000,E1 265.869} C_DIS
LIN {X -0.033,Y -180.915,Z 369.477,A 0.000,B 0.000,C 90.000,E1 265.869} C_DIS
LIN {X -0.003,Y -180.817,Z 369.471,A 0.000,B 0.000,C 90.000,E1 264.837} C_DIS
LIN {X 0.068,Y -178.846,Z 369.442,A 0.000,B 0.000,C 90.000,E1 259.577} C_DIS
LIN {X -0.037,Y -175.889,Z 369.414,A 0.000,B 0.000,C 90.000,E1 254.519} C_DIS
LIN {X 0.070,Y -174.559,Z 369.404,A 0.000,B 0.000,C 90.000,E1 252.779} C_DIS
LIN {X -0.061,Y -171.543,Z 369.381,A 0.000,B 0.000,C 90.000,E1 248.539} C_DIS
LIN {X -0.005,Y -167.768,Z 369.357,A 0.000,B 0.000,C 90.000,E1 244.204} C_DIS
LIN {X -0.064,Y -166.476,Z 369.347,A 0.000,B 0.000,C 90.000,E1 242.487} C_DIS
LIN {X -0.067,Y -163.189,Z 369.328,A 0.000,B 0.000,C 90.000,E1 238.997} C_DIS
LIN {X -0.012,Y -161.150,Z 369.313,A 0.000,B 0.000,C 90.000,E1 236.342} C_DIS
LIN {X 0.024,Y -157.169,Z 369.288,A 0.000,B 0.000,C 90.000,E1 231.904} C_DIS
LIN {X -0.054,Y -155.900,Z 369.279,A 0.000,B 0.000,C 90.000,E1 230.150} C_DIS
LIN {X 0.004,Y -152.149,Z 369.254,A 0.000,B 0.000,C 90.000,E1 225.648} C_DIS
LIN {X 0.023,Y -150.399,Z 369.239,A 0.000,B 0.000,C 90.000,E1 222.933} C_DIS
LIN {X 0.047,Y -147.130,Z 369.213,A 0.000,B 0.000,C 90.000,E1 218.382} C_DIS
LIN {X -0.046,Y -145.692,Z 369.198,A 0.000,B 0.000,C 90.000,E1 215.678} C_DIS
LIN {X 0.036,Y -143.074,Z 369.173,A 0.000,B 0.000,C 90.000,E1 211.052} C_DIS
LIN {X -0.033,Y -141.694,Z 369.152,A 0.000,B 0.000,C 90.000,E1 207.385} C_DIS
LIN {X 0.021,Y -139.463,Z 369.116,A 0.000,B 0.000,C 90.000,E1 200.865} C_DIS
LIN {X -0.056,Y -139.197,Z 369.106,A 0.000,B 0.000,C 90.000,E1 199.033} C_DIS
LIN {X 0.007,Y -138.325,Z 369.054,A 0.000,B 0.000,C 90.000,E1 189.670} C_DIS
LIN {X 0.013,Y -139.449,Z 369.007,A 0.000,B 0.000,C 90.000,E1 181.260} C_DIS
LIN {X -0.048,Y -140.991,Z 368.976,A 0.000,B 0.000,C 90.000,E1 175.698} C_DIS
LIN {X 0.043,Y -142.746,Z 368.955,A 0.000,B 0.000,C 90.000,E1 171.951} C_DIS
LIN {X 0.000,Y -145.143,Z 368.930,A 0.000,B 0.000,C 90.000,E1 167.353} C_DIS
LIN {X -0.007,Y -147.765,Z 368.909,A 0.000,B 0.000,C 90.000,E1 163.685} C_DIS
LIN {X -0.068,Y -150.439,Z 368.889,A 0.000,B 0.000,C 90.000,E1 160.061} C_DIS
LIN {X 0.008,Y -153.885,Z 368.869,A 0.000,B 0.000,C 90.000,E1 156.410} C_DIS
LIN {X 0.002,Y -157.295,Z 368.849,A 0.000,B 0.000,C 90.000,E1 152.820} C_DIS
LIN {X 0.020,Y -161.478,Z 368.829,A 0.000,B 0.000,C 90.000,E1 149.253} C_DIS
LIN {X 0.037,Y -165.677,Z 368.810,A 0.000,B 0.000,C 90.000,E1 145.722} C_DIS
LIN {X -0.076,Y -170.618,Z 368.790,A 0.000,B 0.000,C 90.000,E1 142.271} C_DIS
LIN {X 0.078,Y -175.494,Z 368.771,A 0.000,B 0.000,C 90.000,E1 138.771} C_DIS
LIN {X -0.056,Y -181.115,Z 368.752,A 0.000,B 0.000,C 90.000,E1 135.405} C_DIS
LIN {X 0.072,Y -186.563,Z 368.733,A 0.000,B 0.000,C 90.000,E1 132.000} C_DIS
LIN {X 0.022,Y -191.176,Z 368.720,A 0.000,B 0.000,C 90.000,E1 129.519} C_DIS
LIN {X 0.067,Y -196.982,Z 368.701,A 0.000,B 0.000,C 90.000,E1 126.217} C_DIS
LIN {X -0.028,Y -199.240,Z 368.695,A 0.000,B 0.000,C 90.000,E1 125.105} C_DIS
LIN {X -0.089,Y -298.935,Z 368.695,A 0.000,B 0.000,C 90.000,E1 125.105} C_DIS
LIN {X 0.157,Y -305.231,Z 368.694,A 0.000,B 0.000,C 90.000,E1 124.818} C_DIS
LIN {X -0.020,Y -308.013,Z 368.692,A 0.000,B 0.000,C 90.000,E1 124.612} C_DIS
LIN {X -0.064,Y -311.781,Z 368.689,A 0.000,B 0.000,C 90.000,E1 124.119} C_DIS
LIN {X -0.024,Y -313.499,Z 368.688,A 0.000,B 0.000,C 90.000,E1 123.785} C_DIS
LIN {X 0.018,Y -314.850,Z 368.686,A 0.000,B 0.000,C 90.000,E1 123.452} C_DIS
LIN {X -0.030,Y -326.337,Z 368.668,A 0.000,B 0.000,C 90.000,E1 120.256} C_DIS
LIN {X -0.068,Y -338.081,Z 368.652,A 0.000,B 0.000,C 90.000,E1 117.436} C_DIS
LIN {X 0.068,Y -351.293,Z 368.637,A 0.000,B 0.000,C 90.000,E1 114.643} C_DIS
LIN {X -0.091,Y -364.365,Z 368.624,A 0.000,B 0.000,C 90.000,E1 112.259} C_DIS
LIN {X 0.008,Y -378.785,Z 368.610,A 0.000,B 0.000,C 90.000,E1 109.885} C_DIS
LIN {X -0.001,Y -394.661,Z 368.598,A 0.000,B 0.000,C 90.000,E1 107.583} C_DIS
LIN {X 0.156,Y -412.110,Z 368.585,A 0.000,B 0.000,C 90.000,E1 105.315} C_DIS
LIN {X -0.175,Y -431.254,Z 368.573,A 0.000,B 0.000,C 90.000,E1 103.175} C_DIS
LIN {X -0.189,Y -451.427,Z 368.562,A 0.000,B 0.000,C 90.000,E1 101.130} C_DIS
LIN {X 0.195,Y -472.144,Z 368.551,A 0.000,B 0.000,C 90.000,E1 99.208} C_DIS
LIN {X 0.160,Y -490.635,Z 368.543,A 0.000,B 0.000,C 90.000,E1 97.701} C_DIS
LIN {X -0.166,Y -492.803,Z 368.542,A 0.000,B 0.000,C 90.000,E1 97.530} C_DIS
LIN {X -0.188,Y -494.664,Z 368.540,A 0.000,B 0.000,C 90.000,E1 97.296} C_DIS
LIN {X -0.272,Y -496.072,Z 368.539,A 0.000,B 0.000,C 90.000,E1 97.068} C_DIS
LIN {X -0.017,Y -497.938,Z 368.536,A 0.000,B 0.000,C 90.000,E1 96.549} C_DIS
LIN {X -0.250,Y -498.681,Z 368.534,A 0.000,B 0.000,C 90.000,E1 96.087} C_DIS
LIN {X 0.024,Y -498.426,Z 368.531,A 0.000,B 0.000,C 90.000,E1 95.568} C_DIS
LIN {X -0.196,Y -497.130,Z 368.528,A 0.000,B 0.000,C 90.000,E1 95.106} C_DIS
LIN {X 0.167,Y -496.027,Z 368.527,A 0.000,B 0.000,C 90.000,E1 94.821} C_DIS
LIN {X 0.076,Y -494.540,Z 368.526,A 0.000,B 0.000,C 90.000,E1 94.588} C_DIS
LIN {X 0.183,Y -489.136,Z 368.521,A 0.000,B 0.000,C 90.000,E1 93.841} C_DIS
LIN {X 0.086,Y -481.373,Z 368.516,A 0.000,B 0.000,C 90.000,E1 92.865} C_DIS
LIN {X 0.185,Y -457.746,Z 368.499,A 0.000,B 0.000,C 90.000,E1 89.828} C_DIS
LIN {X -0.128,Y -441.479,Z 368.486,A 0.000,B 0.000,C 90.000,E1 87.535} C_DIS
LIN {X -0.106,Y -423.226,Z 368.470,A 0.000,B 0.000,C 90.000,E1 84.609} C_DIS
LIN {X -0.181,Y -407.948,Z 368.455,A 0.000,B 0.000,C 90.000,E1 81.894} C_DIS
LIN {X 0.146,Y -394.701,Z 368.441,A 0.000,B 0.000,C 90.000,E1 79.342} C_DIS
LIN {X 0.167,Y -384.481,Z 368.430,A 0.000,B 0.000,C 90.000,E1 77.353} C_DIS
LIN {X 0.157,Y -372.804,Z 368.417,A 0.000,B 0.000,C 90.000,E1 75.046} C_DIS
LIN {X -0.028,Y -361.307,Z 368.404,A 0.000,B 0.000,C 90.000,E1 72.725} C_DIS
LIN {X 0.144,Y -351.302,Z 368.392,A 0.000,B 0.000,C 90.000,E1 70.604} C_DIS
LIN {X -0.085,Y -338.680,Z 368.377,A 0.000,B 0.000,C 90.000,E1 67.901} C_DIS
LIN {X -0.017,Y -324.211,Z 368.358,A 0.000,B 0.000,C 90.000,E1 64.460} C_DIS
LIN {X -0.011,Y -313.371,Z 368.342,A 0.000,B 0.000,C 90.000,E1 61.591} C_DIS
LIN {X 0.080,Y -300.960,Z 368.322,A 0.000,B 0.000,C 90.000,E1 57.995} C_DIS
LIN {X 0.014,Y -290.554,Z 368.304,A 0.000,B 0.000,C 90.000,E1 54.689} C_DIS
LIN {X 0.047,Y -282.927,Z 368.289,A 0.000,B 0.000,C 90.000,E1 51.984} C_DIS
LIN {X 0.180,Y -277.367,Z 368.277,A 0.000,B 0.000,C 90.000,E1 49.908} C_DIS
LIN {X -0.004,Y -271.704,Z 368.266,A 0.000,B 0.000,C 90.000,E1 47.877} C_DIS
LIN {X -0.123,Y -266.036,Z 368.254,A 0.000,B 0.000,C 90.000,E1 45.810} C_DIS
LIN {X 0.031,Y -260.311,Z 368.243,A 0.000,B 0.000,C 90.000,E1 43.662} C_DIS
LIN {X 0.070,Y -254.550,Z 368.231,A 0.000,B 0.000,C 90.000,E1 41.515} C_DIS
LIN {X 0.042,Y -248.579,Z 368.219,A 0.000,B 0.000,C 90.000,E1 39.358} C_DIS
LIN {X -0.056,Y -240.726,Z 368.202,A 0.000,B 0.000,C 90.000,E1 36.457} C_DIS
LIN {X -0.102,Y -233.094,Z 368.186,A 0.000,B 0.000,C 90.000,E1 33.499} C_DIS
LIN {X 0.116,Y -223.957,Z 368.165,A 0.000,B 0.000,C 90.000,E1 29.667} C_DIS
LIN {X 0.025,Y -217.290,Z 368.148,A 0.000,B 0.000,C 90.000,E1 26.616} C_DIS
LIN {X -0.031,Y -211.216,Z 368.131,A 0.000,B 0.000,C 90.000,E1 23.515} C_DIS
LIN {X -0.019,Y -205.859,Z 368.113,A 0.000,B 0.000,C 90.000,E1 20.355} C_DIS
LIN {X -0.060,Y -200.019,Z 368.091,A 0.000,B 0.000,C 90.000,E1 16.370} C_DIS
LIN {X 0.001,Y -196.130,Z 368.073,A 0.000,B 0.000,C 90.000,E1 13.119} C_DIS
LIN {X 0.036,Y -192.157,Z 368.050,A 0.000,B 0.000,C 90.000,E1 9.029} C_DIS
LIN {X -0.030,Y -189.456,Z 368.027,A 0.000,B 0.000,C 90.000,E1 4.935} C_DIS
LIN {X 0.069,Y -187.591,Z 367.984,A 0.000,B 0.000,C 90.000,E1 357.020} C_DIS
LIN {X -0.029,Y -189.745,Z 367.938,A 0.000,B 0.000,C 90.000,E1 348.757} C_DIS
LIN {X 0.016,Y -192.932,Z 367.910,A 0.000,B 0.000,C 90.000,E1 343.795} C_DIS
LIN {X 0.022,Y -196.836,Z 367.887,A 0.000,B 0.000,C 90.000,E1 339.699} C_DIS
LIN {X -0.061,Y -201.812,Z 367.865,A 0.000,B 0.000,C 90.000,E1 335.665} C_DIS
LIN {X 0.091,Y -206.643,Z 367.847,A 0.000,B 0.000,C 90.000,E1 332.410} C_DIS
LIN {X 0.039,Y -213.395,Z 367.825,A 0.000,B 0.000,C 90.000,E1 328.456} C_DIS
LIN {X -0.021,Y -220.695,Z 367.803,A 0.000,B 0.000,C 90.000,E1 324.562} C_DIS
LIN {X -0.057,Y -228.965,Z 367.782,A 0.000,B 0.000,C 90.000,E1 320.723} C_DIS
LIN {X -0.031,Y -237.258,Z 367.763,A 0.000,B 0.000,C 90.000,E1 317.310} C_DIS
LIN {X 0.060,Y -246.715,Z 367.744,A 0.000,B 0.000,C 90.000,E1 313.947} C_DIS
LIN {X 0.073,Y -254.934,Z 367.730,A 0.000,B 0.000,C 90.000,E1 311.391} C_DIS
LIN {X -0.071,Y -263.729,Z 367.716,A 0.000,B 0.000,C 90.000,E1 308.910} C_DIS
LIN {X -0.065,Y -274.422,Z 367.700,A 0.000,B 0.000,C 90.000,E1 306.091} C_DIS
LIN {X 0.002,Y -284.178,Z 367.687,A 0.000,B 0.000,C 90.000,E1 303.658} C_DIS
LIN {X 0.123,Y -298.052,Z 367.670,A 0.000,B 0.000,C 90.000,E1 300.590} C_DIS
LIN {X -0.004,Y -311.888,Z 367.655,A 0.000,B 0.000,C 90.000,E1 297.975} C_DIS
LIN {X -0.015,Y -321.281,Z 367.646,A 0.000,B 0.000,C 90.000,E1 296.360} C_DIS
LIN {X 0.020,Y -337.879,Z 367.632,A 0.000,B 0.000,C 90.000,E1 293.823} C_DIS
LIN {X 0.043,Y -353.451,Z 367.620,A 0.000,B 0.000,C 90.000,E1 291.663} C_DIS
LIN {X -0.045,Y -369.414,Z 367.609,A 0.000,B 0.000,C 90.000,E1 289.577} C_DIS
LIN {X 0.137,Y -384.141,Z 367.599,A 0.000,B 0.000,C 90.000,E1 287.819} C_DIS
LIN {X 0.067,Y -401.948,Z 367.588,A 0.000,B 0.000,C 90.000,E1 285.898} C_DIS
LIN {X -0.155,Y -419.882,Z 367.578,A 0.000,B 0.000,C 90.000,E1 284.064} C_DIS
LIN {X -0.019,Y -429.960,Z 367.572,A 0.000,B 0.000,C 90.000,E1 283.008} C_DIS
LIN {X -0.238,Y -437.280,Z 367.568,A 0.000,B 0.000,C 90.000,E1 282.243} C_DIS
LIN {X -0.056,Y -444.212,Z 367.563,A 0.000,B 0.000,C 90.000,E1 281.422} C_DIS
LIN {X 0.188,Y -450.541,Z 367.559,A 0.000,B 0.000,C 90.000,E1 280.602} C_DIS
LIN {X -0.223,Y -458.360,Z 367.553,A 0.000,B 0.000,C 90.000,E1 279.613} C_DIS
LIN {X -0.095,Y -465.487,Z 367.548,A 0.000,B 0.000,C 90.000,E1 278.568} C_DIS
LIN {X 0.055,Y -471.994,Z 367.542,A 0.000,B 0.000,C 90.000,E1 277.530} C_DIS
LIN {X -0.131,Y -477.928,Z 367.536,A 0.000,B 0.000,C 90.000,E1 276.543} C_DIS
LIN {X -0.176,Y -481.956,Z 367.532,A 0.000,B 0.000,C 90.000,E1 275.796} C_DIS
LIN {X -0.011,Y -484.257,Z 367.529,A 0.000,B 0.000,C 90.000,E1 275.277} C_DIS
LIN {X 0.000,Y -486.949,Z 367.525,A 0.000,B 0.000,C 90.000,E1 274.531} C_DIS
LIN {X 0.192,Y -488.319,Z 367.522,A 0.000,B 0.000,C 90.000,E1 274.012} C_DIS
LIN {X -0.129,Y -489.308,Z 367.520,A 0.000,B 0.000,C 90.000,E1 273.555} C_DIS
LIN {X 0.078,Y -489.965,Z 367.517,A 0.000,B 0.000,C 90.000,E1 273.037} C_DIS
LIN {X -0.225,Y -490.299,Z 367.514,A 0.000,B 0.000,C 90.000,E1 272.579} C_DIS
LIN {X -0.033,Y -490.403,Z 367.511,A 0.000,B 0.000,C 90.000,E1 272.064} C_DIS
LIN {X 0.178,Y -490.166,Z 367.509,A 0.000,B 0.000,C 90.000,E1 271.547} C_DIS
LIN {X -0.115,Y -489.628,Z 367.506,A 0.000,B 0.000,C 90.000,E1 271.088} C_DIS
LIN {X 0.081,Y -488.753,Z 367.503,A 0.000,B 0.000,C 90.000,E1 270.573} C_DIS
LIN {X -0.214,Y -487.403,Z 367.500,A 0.000,B 0.000,C 90.000,E1 270.115} C_DIS
LIN {X -0.026,Y -485.527,Z 367.498,A 0.000,B 0.000,C 90.000,E1 269.599} C_DIS
LIN {X -0.179,Y -484.392,Z 367.496,A 0.000,B 0.000,C 90.000,E1 269.370} C_DIS
LIN {X -0.010,Y -481.520,Z 367.494,A 0.000,B 0.000,C 90.000,E1 268.854} C_DIS
LIN {X 0.140,Y -477.868,Z 367.491,A 0.000,B 0.000,C 90.000,E1 268.339} C_DIS
LIN {X -0.189,Y -473.050,Z 367.488,A 0.000,B 0.000,C 90.000,E1 267.879} C_DIS
LIN {X 0.177,Y -467.157,Z 367.485,A 0.000,B 0.000,C 90.000,E1 267.364} C_DIS
LIN {X -0.219,Y -463.878,Z 367.484,A 0.000,B 0.000,C 90.000,E1 267.192} C_DIS
LIN {X 0.106,Y -460.660,Z 367.483,A 0.000,B 0.000,C 90.000,E1 266.963} C_DIS
LIN {X 0.156,Y -453.567,Z 367.481,A 0.000,B 0.000,C 90.000,E1 266.617} C_DIS
LIN {X -0.173,Y -446.213,Z 367.480,A 0.000,B 0.000,C 90.000,E1 266.388} C_DIS
LIN {X -0.042,Y -438.547,Z 367.479,A 0.000,B 0.000,C 90.000,E1 266.159} C_DIS
LIN {X 0.069,Y -429.949,Z 367.478,A 0.000,B 0.000,C 90.000,E1 265.988} C_DIS
LIN {X 0.157,Y -419.510,Z 367.477,A 0.000,B 0.000,C 90.000,E1 265.869} C_DIS
LIN {X 0.002,Y -415.288,Z 367.477,A 0.000,B 0.000,C 90.000,E1 265.869} C_DIS
LIN {X -0.032,Y -180.915,Z 367.477,A 0.000,B 0.000,C 90.000,E1 265.869} C_DIS
LIN {X -0.003,Y -180.817,Z 367.471,A 0.000,B 0.000,C 90.000,E1 264.837} C_DIS
LIN {X 0.067,Y -178.846,Z 367.442,A 0.000,B 0.000,C 90.000,E1 259.577} C_DIS
LIN {X -0.038,Y -175.890,Z 367.414,A 0.000,B 0.000,C 90.000,E1 254.519} C_DIS
LIN {X 0.069,Y -174.559,Z 367.404,A 0.000,B 0.000,C 90.000,E1 252.779} C_DIS
LIN {X -0.062,Y -171.542,Z 367.381,A 0.000,B 0.000,C 90.000,E1 248.539} C_DIS
LIN {X -0.006,Y -167.767,Z 367.357,A 0.000,B 0.000,C 90.000,E1 244.204} C_DIS
LIN {X -0.064,Y -166.476,Z 367.347,A 0.000,B 0.000,C 90.000,E1 242.487} C_DIS
LIN {X -0.067,Y -163.189,Z 367.328,A 0.000,B 0.000,C 90.000,E1 238.997} C_DIS
LIN {X -0.012,Y -161.150,Z 367.313,A 0.000,B 0.000,C 90.000,E1 236.342} C_DIS
LIN {X 0.023,Y -157.168,Z 367.288,A 0.000,B 0.000,C 90.000,E1 231.904} C_DIS
LIN {X -0.054,Y -155.900,Z 367.279,A 0.000,B 0.000,C 90.000,E1 230.150} C_DIS
LIN {X 0.004,Y -152.149,Z 367.254,A 0.000,B 0.000,C 90.000,E1 225.648} C_DIS
LIN {X 0.023,Y -150.399,Z 367.239,A 0.000,B 0.000,C 90.000,E1 222.933} C_DIS
LIN {X 0.047,Y -147.129,Z 367.213,A 0.000,B 0.000,C 90.000,E1 218.382} C_DIS
LIN {X 0.038,Y -145.691,Z 367.198,A 0.000,B 0.000,C 90.000,E1 215.644} C_DIS
LIN {X 0.035,Y -143.074,Z 367.173,A 0.000,B 0.000,C 90.000,E1 211.052} C_DIS
LIN {X -0.034,Y -141.693,Z 367.152,A 0.000,B 0.000,C 90.000,E1 207.385} C_DIS
LIN {X 0.020,Y -139.463,Z 367.116,A 0.000,B 0.000,C 90.000,E1 200.865} C_DIS
LIN {X -0.056,Y -139.197,Z 367.106,A 0.000,B 0.000,C 90.000,E1 199.033} C_DIS
LIN {X 0.007,Y -138.326,Z 367.054,A 0.000,B 0.000,C 90.000,E1 189.670} C_DIS
LIN {X 0.012,Y -139.449,Z 367.007,A 0.000,B 0.000,C 90.000,E1 181.260} C_DIS
LIN {X -0.048,Y -140.992,Z 366.976,A 0.000,B 0.000,C 90.000,E1 175.698} C_DIS
LIN {X 0.043,Y -142.746,Z 366.955,A 0.000,B 0.000,C 90.000,E1 171.951} C_DIS
LIN {X -0.001,Y -145.143,Z 366.930,A 0.000,B 0.000,C 90.000,E1 167.353} C_DIS
LIN {X -0.008,Y -147.766,Z 366.909,A 0.000,B 0.000,C 90.000,E1 163.685} C_DIS
LIN {X -0.069,Y -150.440,Z 366.889,A 0.000,B 0.000,C 90.000,E1 160.061} C_DIS
LIN {X 0.007,Y -153.885,Z 366.869,A 0.000,B 0.000,C 90.000,E1 156.410} C_DIS
LIN {X 0.001,Y -157.295,Z 366.849,A 0.000,B 0.000,C 90.000,E1 152.820} C_DIS
LIN {X 0.019,Y -161.478,Z 366.829,A 0.000,B 0.000,C 90.000,E1 149.253} C_DIS
LIN {X 0.036,Y -165.678,Z 366.810,A 0.000,B 0.000,C 90.000,E1 145.722} C_DIS
LIN {X -0.076,Y -170.618,Z 366.790,A 0.000,B 0.000,C 90.000,E1 142.271} C_DIS
LIN {X 0.077,Y -175.494,Z 366.771,A 0.000,B 0.000,C 90.000,E1 138.771} C_DIS
LIN {X -0.056,Y -181.115,Z 366.752,A 0.000,B 0.000,C 90.000,E1 135.405} C_DIS
LIN {X 0.072,Y -186.563,Z 366.733,A 0.000,B 0.000,C 90.000,E1 132.000} C_DIS
LIN {X 0.021,Y -191.176,Z 366.720,A 0.000,B 0.000,C 90.000,E1 129.519} C_DIS
LIN {X 0.067,Y -196.982,Z 366.701,A 0.000,B 0.000,C 90.000,E1 126.217} C_DIS
LIN {X 0.061,Y -199.352,Z 366.695,A 0.000,B 0.000,C 90.000,E1 125.025} C_DIS
LIN {X 0.046,Y -298.734,Z 366.695,A 0.000,B 0.000,C 90.000,E1 125.025} C_DIS
LIN {X 0.001,Y -299.709,Z 366.695,A 0.000,B 0.000,C 90.000,E1 125.025} C_DIS
LIN {X -0.010,Y -305.037,Z 366.693,A 0.000,B 0.000,C 90.000,E1 124.818} C_DIS
LIN {X -0.022,Y -307.624,Z 366.692,A 0.000,B 0.000,C 90.000,E1 124.612} C_DIS
LIN {X 0.081,Y -311.440,Z 366.690,A 0.000,B 0.000,C 90.000,E1 124.119} C_DIS
LIN {X 0.120,Y -313.271,Z 366.688,A 0.000,B 0.000,C 90.000,E1 123.785} C_DIS
LIN {X -0.101,Y -314.707,Z 366.686,A 0.000,B 0.000,C 90.000,E1 123.499} C_DIS
LIN {X 0.051,Y -327.451,Z 366.666,A 0.000,B 0.000,C 90.000,E1 119.951} C_DIS
LIN {X 0.054,Y -339.342,Z 366.651,A 0.000,B 0.000,C 90.000,E1 117.129} C_DIS
LIN {X -0.076,Y -352.706,Z 366.635,A 0.000,B 0.000,C 90.000,E1 114.387} C_DIS
LIN {X -0.007,Y -365.928,Z 366.622,A 0.000,B 0.000,C 90.000,E1 111.972} C_DIS
LIN {X -0.080,Y -380.510,Z 366.609,A 0.000,B 0.000,C 90.000,E1 109.631} C_DIS
LIN {X -0.058,Y -396.560,Z 366.596,A 0.000,B 0.000,C 90.000,E1 107.330} C_DIS
LIN {X 0.132,Y -414.197,Z 366.584,A 0.000,B 0.000,C 90.000,E1 105.064} C_DIS
LIN {X 0.188,Y -433.509,Z 366.572,A 0.000,B 0.000,C 90.000,E1 102.883} C_DIS
LIN {X -0.091,Y -453.748,Z 366.560,A 0.000,B 0.000,C 90.000,E1 100.894} C_DIS
LIN {X -0.022,Y -474.524,Z 366.550,A 0.000,B 0.000,C 90.000,E1 99.029} C_DIS
LIN {X -0.192,Y -490.416,Z 366.543,A 0.000,B 0.000,C 90.000,E1 97.757} C_DIS
LIN {X -0.033,Y -492.694,Z 366.542,A 0.000,B 0.000,C 90.000,E1 97.530} C_DIS
LIN {X 0.006,Y -494.583,Z 366.541,A 0.000,B 0.000,C 90.000,E1 97.296} C_DIS
LIN {X -0.019,Y -496.023,Z 366.539,A 0.000,B 0.000,C 90.000,E1 97.068} C_DIS
LIN {X -0.259,Y -498.013,Z 366.537,A 0.000,B 0.000,C 90.000,E1 96.606} C_DIS
LIN {X 0.004,Y -498.857,Z 366.534,A 0.000,B 0.000,C 90.000,E1 96.087} C_DIS
LIN {X -0.218,Y -498.697,Z 366.531,A 0.000,B 0.000,C 90.000,E1 95.625} C_DIS
LIN {X 0.059,Y -497.507,Z 366.528,A 0.000,B 0.000,C 90.000,E1 95.106} C_DIS
LIN {X -0.073,Y -496.467,Z 366.527,A 0.000,B 0.000,C 90.000,E1 94.878} C_DIS
LIN {X -0.162,Y -495.060,Z 366.526,A 0.000,B 0.000,C 90.000,E1 94.645} C_DIS
LIN {X -0.048,Y -489.702,Z 366.522,A 0.000,B 0.000,C 90.000,E1 93.898} C_DIS
LIN {X -0.136,Y -481.953,Z 366.516,A 0.000,B 0.000,C 90.000,E1 92.922} C_DIS
LIN {X 0.207,Y -460.184,Z 366.501,A 0.000,B 0.000,C 90.000,E1 90.115} C_DIS
LIN {X -0.053,Y -443.703,Z 366.488,A 0.000,B 0.000,C 90.000,E1 87.822} C_DIS
LIN {X 0.166,Y -423.665,Z 366.470,A 0.000,B 0.000,C 90.000,E1 84.609} C_DIS
LIN {X 0.094,Y -408.381,Z 366.455,A 0.000,B 0.000,C 90.000,E1 81.894} C_DIS
LIN {X 0.036,Y -395.150,Z 366.441,A 0.000,B 0.000,C 90.000,E1 79.398} C_DIS
LIN {X 0.070,Y -384.930,Z 366.430,A 0.000,B 0.000,C 90.000,E1 77.409} C_DIS
LIN {X 0.083,Y -371.826,Z 366.416,A 0.000,B 0.000,C 90.000,E1 74.810} C_DIS
LIN {X -0.089,Y -361.748,Z 366.404,A 0.000,B 0.000,C 90.000,E1 72.779} C_DIS
LIN {X -0.019,Y -351.708,Z 366.393,A 0.000,B 0.000,C 90.000,E1 70.678} C_DIS
LIN {X 0.073,Y -339.035,Z 366.377,A 0.000,B 0.000,C 90.000,E1 67.922} C_DIS
LIN {X -0.166,Y -324.528,Z 366.358,A 0.000,B 0.000,C 90.000,E1 64.537} C_DIS
LIN {X -0.003,Y -313.689,Z 366.342,A 0.000,B 0.000,C 90.000,E1 61.641} C_DIS
LIN {X -0.052,Y -301.274,Z 366.323,A 0.000,B 0.000,C 90.000,E1 58.074} C_DIS
LIN {X -0.109,Y -290.840,Z 366.304,A 0.000,B 0.000,C 90.000,E1 54.769} C_DIS
LIN {X -0.068,Y -283.215,Z 366.289,A 0.000,B 0.000,C 90.000,E1 52.065} C_DIS
LIN {X 0.083,Y -275.764,Z 366.274,A 0.000,B 0.000,C 90.000,E1 49.299} C_DIS
LIN {X 0.019,Y -268.184,Z 366.259,A 0.000,B 0.000,C 90.000,E1 46.539} C_DIS
LIN {X 0.121,Y -260.588,Z 366.243,A 0.000,B 0.000,C 90.000,E1 43.704} C_DIS
LIN {X -0.012,Y -254.836,Z 366.231,A 0.000,B 0.000,C 90.000,E1 41.595} C_DIS
LIN {X -0.032,Y -248.905,Z 366.219,A 0.000,B 0.000,C 90.000,E1 39.439} C_DIS
LIN {X 0.026,Y -241.043,Z 366.203,A 0.000,B 0.000,C 90.000,E1 36.503} C_DIS
LIN {X -0.152,Y -233.398,Z 366.186,A 0.000,B 0.000,C 90.000,E1 33.579} C_DIS
LIN {X 0.083,Y -224.219,Z 366.165,A 0.000,B 0.000,C 90.000,E1 29.745} C_DIS
LIN {X 0.004,Y -217.546,Z 366.148,A 0.000,B 0.000,C 90.000,E1 26.693} C_DIS
LIN {X 0.045,Y -211.428,Z 366.131,A 0.000,B 0.000,C 90.000,E1 23.567} C_DIS
LIN {X -0.016,Y -206.034,Z 366.113,A 0.000,B 0.000,C 90.000,E1 20.429} C_DIS
LIN {X -0.043,Y -200.174,Z 366.091,A 0.000,B 0.000,C 90.000,E1 16.441} C_DIS
LIN {X 0.074,Y -196.261,Z 366.073,A 0.000,B 0.000,C 90.000,E1 13.175} C_DIS
LIN {X 0.079,Y -192.248,Z 366.051,A 0.000,B 0.000,C 90.000,E1 9.095} C_DIS
LIN {X 0.042,Y -189.513,Z 366.028,A 0.000,B 0.000,C 90.000,E1 4.992} C_DIS
LIN {X 0.069,Y -187.560,Z 365.984,A 0.000,B 0.000,C 90.000,E1 357.020} C_DIS
LIN {X -0.031,Y -189.716,Z 365.938,A 0.000,B 0.000,C 90.000,E1 348.757} C_DIS
LIN {X 0.012,Y -192.878,Z 365.910,A 0.000,B 0.000,C 90.000,E1 343.795} C_DIS
LIN {X 0.016,Y -196.772,Z 365.887,A 0.000,B 0.000,C 90.000,E1 339.699} C_DIS
LIN {X -0.069,Y -201.744,Z 365.865,A 0.000,B 0.000,C 90.000,E1 335.665} C_DIS
LIN {X 0.081,Y -206.556,Z 365.847,A 0.000,B 0.000,C 90.000,E1 332.410} C_DIS
LIN {X 0.026,Y -213.300,Z 365.825,A 0.000,B 0.000,C 90.000,E1 328.456} C_DIS
LIN {X -0.037,Y -220.597,Z 365.803,A 0.000,B 0.000,C 90.000,E1 324.562} C_DIS
LIN {X -0.076,Y -228.863,Z 365.782,A 0.000,B 0.000,C 90.000,E1 320.723} C_DIS
LIN {X -0.016,Y -236.194,Z 365.765,A 0.000,B 0.000,C 90.000,E1 317.676} C_DIS
LIN {X -0.123,Y -245.532,Z 365.746,A 0.000,B 0.000,C 90.000,E1 314.352} C_DIS
LIN {X 0.044,Y -254.879,Z 365.730,A 0.000,B 0.000,C 90.000,E1 311.391} C_DIS
LIN {X -0.102,Y -263.656,Z 365.716,A 0.000,B 0.000,C 90.000,E1 308.910} C_DIS
LIN {X -0.100,Y -274.348,Z 365.700,A 0.000,B 0.000,C 90.000,E1 306.091} C_DIS
LIN {X 0.079,Y -285.660,Z 365.685,A 0.000,B 0.000,C 90.000,E1 303.293} C_DIS
LIN {X 0.084,Y -298.106,Z 365.670,A 0.000,B 0.000,C 90.000,E1 300.590} C_DIS
LIN {X 0.005,Y -313.826,Z 365.654,A 0.000,B 0.000,C 90.000,E1 297.641} C_DIS
LIN {X 0.016,Y -323.471,Z 365.645,A 0.000,B 0.000,C 90.000,E1 296.027} C_DIS
LIN {X -0.035,Y -340.304,Z 365.631,A 0.000,B 0.000,C 90.000,E1 293.515} C_DIS
LIN {X 0.011,Y -353.679,Z 365.620,A 0.000,B 0.000,C 90.000,E1 291.663} C_DIS
LIN {X 0.142,Y -371.939,Z 365.607,A 0.000,B 0.000,C 90.000,E1 289.268} C_DIS
LIN {X 0.174,Y -396.968,Z 365.591,A 0.000,B 0.000,C 90.000,E1 286.441} C_DIS
LIN {X -0.038,Y -414.782,Z 365.581,A 0.000,B 0.000,C 90.000,E1 284.592} C_DIS
LIN {X -0.149,Y -427.543,Z 365.574,A 0.000,B 0.000,C 90.000,E1 283.300} C_DIS
LIN {X 0.096,Y -434.905,Z 365.569,A 0.000,B 0.000,C 90.000,E1 282.479} C_DIS
LIN {X -0.175,Y -441.947,Z 365.565,A 0.000,B 0.000,C 90.000,E1 281.715} C_DIS
LIN {X 0.052,Y -448.439,Z 365.561,A 0.000,B 0.000,C 90.000,E1 280.894} C_DIS
LIN {X 0.066,Y -456.403,Z 365.555,A 0.000,B 0.000,C 90.000,E1 279.849} C_DIS
LIN {X 0.178,Y -463.682,Z 365.549,A 0.000,B 0.000,C 90.000,E1 278.803} C_DIS
LIN {X 0.067,Y -468.683,Z 365.545,A 0.000,B 0.000,C 90.000,E1 278.049} C_DIS
LIN {X -0.210,Y -474.908,Z 365.539,A 0.000,B 0.000,C 90.000,E1 277.068} C_DIS
LIN {X -0.226,Y -479.201,Z 365.535,A 0.000,B 0.000,C 90.000,E1 276.315} C_DIS
LIN {X 0.218,Y -482.982,Z 365.531,A 0.000,B 0.000,C 90.000,E1 275.511} C_DIS
LIN {X -0.088,Y -485.103,Z 365.528,A 0.000,B 0.000,C 90.000,E1 275.049} C_DIS
LIN {X 0.098,Y -486.839,Z 365.525,A 0.000,B 0.000,C 90.000,E1 274.531} C_DIS
LIN {X -0.198,Y -488.193,Z 365.522,A 0.000,B 0.000,C 90.000,E1 274.069} C_DIS
LIN {X -0.031,Y -489.162,Z 365.520,A 0.000,B 0.000,C 90.000,E1 273.555} C_DIS
LIN {X 0.174,Y -489.807,Z 365.517,A 0.000,B 0.000,C 90.000,E1 273.037} C_DIS
LIN {X -0.130,Y -490.120,Z 365.514,A 0.000,B 0.000,C 90.000,E1 272.579} C_DIS
LIN {X 0.062,Y -490.192,Z 365.512,A 0.000,B 0.000,C 90.000,E1 272.064} C_DIS
LIN {X -0.218,Y -489.966,Z 365.509,A 0.000,B 0.000,C 90.000,E1 271.604} C_DIS
LIN {X -0.023,Y -489.420,Z 365.506,A 0.000,B 0.000,C 90.000,E1 271.088} C_DIS
LIN {X 0.171,Y -488.528,Z 365.503,A 0.000,B 0.000,C 90.000,E1 270.573} C_DIS
LIN {X -0.124,Y -487.210,Z 365.501,A 0.000,B 0.000,C 90.000,E1 270.115} C_DIS
LIN {X 0.062,Y -485.374,Z 365.498,A 0.000,B 0.000,C 90.000,E1 269.599} C_DIS
LIN {X -0.092,Y -484.275,Z 365.496,A 0.000,B 0.000,C 90.000,E1 269.370} C_DIS
LIN {X 0.076,Y -481.453,Z 365.494,A 0.000,B 0.000,C 90.000,E1 268.854} C_DIS
LIN {X 0.225,Y -477.820,Z 365.491,A 0.000,B 0.000,C 90.000,E1 268.339} C_DIS
LIN {X 0.071,Y -475.626,Z 365.490,A 0.000,B 0.000,C 90.000,E1 268.108} C_DIS
LIN {X 0.190,Y -470.241,Z 365.487,A 0.000,B 0.000,C 90.000,E1 267.593} C_DIS
LIN {X 0.185,Y -467.233,Z 365.485,A 0.000,B 0.000,C 90.000,E1 267.364} C_DIS
LIN {X 0.179,Y -463.834,Z 365.484,A 0.000,B 0.000,C 90.000,E1 267.135} C_DIS
LIN {X 0.035,Y -460.641,Z 365.483,A 0.000,B 0.000,C 90.000,E1 266.963} C_DIS
LIN {X 0.069,Y -453.579,Z 365.481,A 0.000,B 0.000,C 90.000,E1 266.617} C_DIS
LIN {X 0.180,Y -446.172,Z 365.480,A 0.000,B 0.000,C 90.000,E1 266.331} C_DIS
LIN {X -0.133,Y -438.564,Z 365.479,A 0.000,B 0.000,C 90.000,E1 266.159} C_DIS
LIN {X -0.017,Y -429.797,Z 365.478,A 0.000,B 0.000,C 90.000,E1 265.988} C_DIS
LIN {X 0.078,Y -419.202,Z 365.477,A 0.000,B 0.000,C 90.000,E1 265.869} C_DIS
LIN {X -0.076,Y -414.405,Z 365.477,A 0.000,B 0.000,C 90.000,E1 265.869} C_DIS
LIN {X -0.067,Y -180.915,Z 365.477,A 0.000,B 0.000,C 90.000,E1 265.869} C_DIS
LIN {X -0.038,Y -180.813,Z 365.471,A 0.000,B 0.000,C 90.000,E1 264.837} C_DIS
LIN {X 0.032,Y -178.840,Z 365.442,A 0.000,B 0.000,C 90.000,E1 259.577} C_DIS
LIN {X -0.071,Y -175.884,Z 365.414,A 0.000,B 0.000,C 90.000,E1 254.519} C_DIS
LIN {X 0.035,Y -174.549,Z 365.404,A 0.000,B 0.000,C 90.000,E1 252.779} C_DIS
LIN {X -0.032,Y -171.534,Z 365.381,A 0.000,B 0.000,C 90.000,E1 248.518} C_DIS
LIN {X -0.038,Y -167.759,Z 365.357,A 0.000,B 0.000,C 90.000,E1 244.204} C_DIS
LIN {X -0.096,Y -166.465,Z 365.347,A 0.000,B 0.000,C 90.000,E1 242.487} C_DIS
LIN {X 0.040,Y -163.179,Z 365.328,A 0.000,B 0.000,C 90.000,E1 238.948} C_DIS
LIN {X -0.045,Y -161.140,Z 365.313,A 0.000,B 0.000,C 90.000,E1 236.342} C_DIS
LIN {X -0.008,Y -157.160,Z 365.288,A 0.000,B 0.000,C 90.000,E1 231.904} C_DIS
LIN {X 0.015,Y -155.892,Z 365.278,A 0.000,B 0.000,C 90.000,E1 230.114} C_DIS
LIN {X -0.028,Y -152.141,Z 365.254,A 0.000,B 0.000,C 90.000,E1 225.648} C_DIS
LIN {X -0.007,Y -150.391,Z 365.238,A 0.000,B 0.000,C 90.000,E1 222.933} C_DIS
LIN {X 0.017,Y -147.122,Z 365.213,A 0.000,B 0.000,C 90.000,E1 218.382} C_DIS
LIN {X 0.008,Y -145.687,Z 365.198,A 0.000,B 0.000,C 90.000,E1 215.644} C_DIS
LIN {X 0.005,Y -143.069,Z 365.173,A 0.000,B 0.000,C 90.000,E1 211.052} C_DIS
LIN {X -0.063,Y -141.689,Z 365.152,A 0.000,B 0.000,C 90.000,E1 207.385} C_DIS
LIN {X -0.009,Y -139.461,Z 365.116,A 0.000,B 0.000,C 90.000,E1 200.865} C_DIS
LIN {X -0.041,Y -139.195,Z 365.106,A 0.000,B 0.000,C 90.000,E1 199.014} C_DIS
LIN {X -0.022,Y -138.325,Z 365.054,A 0.000,B 0.000,C 90.000,E1 189.670} C_DIS
LIN {X -0.017,Y -139.451,Z 365.007,A 0.000,B 0.000,C 90.000,E1 181.260} C_DIS
LIN {X 0.063,Y -140.996,Z 364.976,A 0.000,B 0.000,C 90.000,E1 175.641} C_DIS
LIN {X 0.013,Y -142.750,Z 364.955,A 0.000,B 0.000,C 90.000,E1 171.951} C_DIS
LIN {X -0.031,Y -145.150,Z 364.930,A 0.000,B 0.000,C 90.000,E1 167.353} C_DIS
LIN {X -0.038,Y -147.773,Z 364.909,A 0.000,B 0.000,C 90.000,E1 163.685} C_DIS
LIN {X 0.042,Y -150.450,Z 364.889,A 0.000,B 0.000,C 90.000,E1 160.007} C_DIS
LIN {X -0.024,Y -153.896,Z 364.869,A 0.000,B 0.000,C 90.000,E1 156.410} C_DIS
LIN {X 0.041,Y -157.307,Z 364.849,A 0.000,B 0.000,C 90.000,E1 152.794} C_DIS
LIN {X -0.012,Y -161.494,Z 364.829,A 0.000,B 0.000,C 90.000,E1 149.253} C_DIS
LIN {X 0.004,Y -165.693,Z 364.810,A 0.000,B 0.000,C 90.000,E1 145.722} C_DIS
LIN {X -0.109,Y -170.636,Z 364.790,A 0.000,B 0.000,C 90.000,E1 142.271} C_DIS
LIN {X 0.043,Y -175.511,Z 364.771,A 0.000,B 0.000,C 90.000,E1 138.771} C_DIS
LIN {X -0.091,Y -181.131,Z 364.752,A 0.000,B 0.000,C 90.000,E1 135.405} C_DIS
LIN {X 0.036,Y -186.581,Z 364.733,A 0.000,B 0.000,C 90.000,E1 132.000} C_DIS
LIN {X -0.014,Y -191.194,Z 364.720,A 0.000,B 0.000,C 90.000,E1 129.519} C_DIS
LIN {X 0.031,Y -197.003,Z 364.701,A 0.000,B 0.000,C 90.000,E1 126.217} C_DIS
LIN {X 0.009,Y -199.478,Z 364.694,A 0.000,B 0.000,C 90.000,E1 124.978} C_DIS
LIN {X -0.023,Y -299.641,Z 364.694,A 0.000,B 0.000,C 90.000,E1 124.978} C_DIS
LIN {X 0.040,Y -304.944,Z 364.693,A 0.000,B 0.000,C 90.000,E1 124.771} C_DIS
LIN {X -0.078,Y -307.316,Z 364.692,A 0.000,B 0.000,C 90.000,E1 124.612} C_DIS
LIN {X 0.137,Y -311.177,Z 364.690,A 0.000,B 0.000,C 90.000,E1 124.119} C_DIS
LIN {X -0.032,Y -313.056,Z 364.688,A 0.000,B 0.000,C 90.000,E1 123.833} C_DIS
LIN {X 0.059,Y -314.532,Z 364.686,A 0.000,B 0.000,C 90.000,E1 123.499} C_DIS
LIN {X -0.072,Y -327.318,Z 364.667,A 0.000,B 0.000,C 90.000,E1 120.001} C_DIS
LIN {X -0.085,Y -339.195,Z 364.651,A 0.000,B 0.000,C 90.000,E1 117.180} C_DIS
LIN {X 0.090,Y -352.545,Z 364.636,A 0.000,B 0.000,C 90.000,E1 114.387} C_DIS
LIN {X -0.179,Y -365.751,Z 364.622,A 0.000,B 0.000,C 90.000,E1 112.025} C_DIS
LIN {X 0.089,Y -380.317,Z 364.609,A 0.000,B 0.000,C 90.000,E1 109.631} C_DIS
LIN {X 0.114,Y -396.350,Z 364.596,A 0.000,B 0.000,C 90.000,E1 107.330} C_DIS
LIN {X -0.202,Y -413.968,Z 364.584,A 0.000,B 0.000,C 90.000,E1 105.134} C_DIS
LIN {X -0.062,Y -433.267,Z 364.572,A 0.000,B 0.000,C 90.000,E1 102.939} C_DIS
LIN {X 0.074,Y -453.499,Z 364.561,A 0.000,B 0.000,C 90.000,E1 100.894} C_DIS
LIN {X 0.134,Y -474.269,Z 364.550,A 0.000,B 0.000,C 90.000,E1 99.029} C_DIS
LIN {X -0.040,Y -490.157,Z 364.543,A 0.000,B 0.000,C 90.000,E1 97.757} C_DIS
LIN {X 0.118,Y -492.551,Z 364.542,A 0.000,B 0.000,C 90.000,E1 97.530} C_DIS
LIN {X 0.217,Y -494.475,Z 364.541,A 0.000,B 0.000,C 90.000,E1 97.296} C_DIS
LIN {X -0.240,Y -495.947,Z 364.539,A 0.000,B 0.000,C 90.000,E1 97.125} C_DIS
LIN {X 0.163,Y -497.173,Z 364.538,A 0.000,B 0.000,C 90.000,E1 96.834} C_DIS
LIN {X 0.013,Y -498.067,Z 364.537,A 0.000,B 0.000,C 90.000,E1 96.606} C_DIS
LIN {X -0.213,Y -499.011,Z 364.534,A 0.000,B 0.000,C 90.000,E1 96.144} C_DIS
LIN {X 0.060,Y -498.949,Z 364.531,A 0.000,B 0.000,C 90.000,E1 95.625} C_DIS
LIN {X -0.157,Y -497.867,Z 364.529,A 0.000,B 0.000,C 90.000,E1 95.163} C_DIS
LIN {X 0.207,Y -496.892,Z 364.527,A 0.000,B 0.000,C 90.000,E1 94.878} C_DIS
LIN {X 0.118,Y -495.566,Z 364.526,A 0.000,B 0.000,C 90.000,E1 94.645} C_DIS
LIN {X 0.232,Y -490.289,Z 364.522,A 0.000,B 0.000,C 90.000,E1 93.898} C_DIS
LIN {X 0.147,Y -482.550,Z 364.516,A 0.000,B 0.000,C 90.000,E1 92.922} C_DIS
LIN {X 0.035,Y -460.750,Z 364.501,A 0.000,B 0.000,C 90.000,E1 90.172} C_DIS
LIN {X -0.205,Y -444.219,Z 364.488,A 0.000,B 0.000,C 90.000,E1 87.879} C_DIS
LIN {X 0.040,Y -424.126,Z 364.470,A 0.000,B 0.000,C 90.000,E1 84.666} C_DIS
LIN {X 0.105,Y -407.342,Z 364.454,A 0.000,B 0.000,C 90.000,E1 81.659} C_DIS
LIN {X -0.053,Y -395.623,Z 364.441,A 0.000,B 0.000,C 90.000,E1 79.454} C_DIS
LIN {X -0.003,Y -385.391,Z 364.430,A 0.000,B 0.000,C 90.000,E1 77.465} C_DIS
LIN {X 0.028,Y -372.302,Z 364.416,A 0.000,B 0.000,C 90.000,E1 74.866} C_DIS
LIN {X -0.164,Y -360.761,Z 364.403,A 0.000,B 0.000,C 90.000,E1 72.543} C_DIS
LIN {X -0.004,Y -350.701,Z 364.391,A 0.000,B 0.000,C 90.000,E1 70.423} C_DIS
LIN {X 0.071,Y -338.032,Z 364.376,A 0.000,B 0.000,C 90.000,E1 67.667} C_DIS
LIN {X 0.092,Y -323.626,Z 364.357,A 0.000,B 0.000,C 90.000,E1 64.229} C_DIS
LIN {X -0.056,Y -312.849,Z 364.341,A 0.000,B 0.000,C 90.000,E1 61.385} C_DIS
LIN {X -0.005,Y -301.601,Z 364.323,A 0.000,B 0.000,C 90.000,E1 58.122} C_DIS
LIN {X -0.045,Y -291.145,Z 364.304,A 0.000,B 0.000,C 90.000,E1 54.815} C_DIS
LIN {X 0.010,Y -283.507,Z 364.290,A 0.000,B 0.000,C 90.000,E1 52.110} C_DIS
LIN {X -0.004,Y -276.048,Z 364.274,A 0.000,B 0.000,C 90.000,E1 49.380} C_DIS
LIN {X -0.028,Y -270.360,Z 364.263,A 0.000,B 0.000,C 90.000,E1 47.310} C_DIS
LIN {X -0.051,Y -262.768,Z 364.247,A 0.000,B 0.000,C 90.000,E1 44.514} C_DIS
LIN {X 0.037,Y -257.064,Z 364.235,A 0.000,B 0.000,C 90.000,E1 42.366} C_DIS
LIN {X 0.027,Y -251.211,Z 364.223,A 0.000,B 0.000,C 90.000,E1 40.216} C_DIS
LIN {X 0.127,Y -245.296,Z 364.211,A 0.000,B 0.000,C 90.000,E1 38.016} C_DIS
LIN {X -0.009,Y -237.507,Z 364.195,A 0.000,B 0.000,C 90.000,E1 35.105} C_DIS
LIN {X -0.079,Y -229.952,Z 364.178,A 0.000,B 0.000,C 90.000,E1 32.133} C_DIS
LIN {X 0.002,Y -222.760,Z 364.162,A 0.000,B 0.000,C 90.000,E1 29.077} C_DIS
LIN {X 0.077,Y -216.230,Z 364.144,A 0.000,B 0.000,C 90.000,E1 25.976} C_DIS
LIN {X -0.092,Y -210.231,Z 364.127,A 0.000,B 0.000,C 90.000,E1 22.898} C_DIS
LIN {X 0.018,Y -204.981,Z 364.109,A 0.000,B 0.000,C 90.000,E1 19.704} C_DIS
LIN {X -0.042,Y -199.268,Z 364.087,A 0.000,B 0.000,C 90.000,E1 15.717} C_DIS
LIN {X -0.020,Y -194.685,Z 364.065,A 0.000,B 0.000,C 90.000,E1 11.658} C_DIS
LIN {X -0.090,Y -191.076,Z 364.042,A 0.000,B 0.000,C 90.000,E1 7.587} C_DIS
LIN {X 0.020,Y -188.223,Z 364.010,A 0.000,B 0.000,C 90.000,E1 1.776} C_DIS
LIN {X 0.051,Y -188.149,Z 363.961,A 0.000,B 0.000,C 90.000,E1 352.875} C_DIS
LIN {X -0.049,Y -191.063,Z 363.924,A 0.000,B 0.000,C 90.000,E1 346.284} C_DIS
LIN {X -0.086,Y -194.265,Z 363.901,A 0.000,B 0.000,C 90.000,E1 342.181} C_DIS
LIN {X -0.100,Y -198.591,Z 363.878,A 0.000,B 0.000,C 90.000,E1 338.103} C_DIS
LIN {X 0.031,Y -203.975,Z 363.856,A 0.000,B 0.000,C 90.000,E1 334.024} C_DIS
LIN {X -0.028,Y -210.440,Z 363.834,A 0.000,B 0.000,C 90.000,E1 330.049} C_DIS
LIN {X -0.094,Y -216.031,Z 363.816,A 0.000,B 0.000,C 90.000,E1 326.914} C_DIS
LIN {X -0.036,Y -222.105,Z 363.799,A 0.000,B 0.000,C 90.000,E1 323.783} C_DIS
LIN {X 0.116,Y -230.529,Z 363.777,A 0.000,B 0.000,C 90.000,E1 319.908} C_DIS
LIN {X 0.015,Y -239.135,Z 363.759,A 0.000,B 0.000,C 90.000,E1 316.539} C_DIS
LIN {X -0.011,Y -248.848,Z 363.740,A 0.000,B 0.000,C 90.000,E1 313.218} C_DIS
LIN {X 0.108,Y -259.811,Z 363.722,A 0.000,B 0.000,C 90.000,E1 309.930} C_DIS
LIN {X -0.128,Y -271.564,Z 363.704,A 0.000,B 0.000,C 90.000,E1 306.790} C_DIS
LIN {X -0.068,Y -284.163,Z 363.687,A 0.000,B 0.000,C 90.000,E1 303.658} C_DIS
LIN {X 0.050,Y -298.180,Z 363.670,A 0.000,B 0.000,C 90.000,E1 300.590} C_DIS
LIN {X -0.077,Y -312.125,Z 363.655,A 0.000,B 0.000,C 90.000,E1 297.975} C_DIS
LIN {X -0.086,Y -321.652,Z 363.646,A 0.000,B 0.000,C 90.000,E1 296.360} C_DIS
LIN {X -0.044,Y -338.327,Z 363.632,A 0.000,B 0.000,C 90.000,E1 293.823} C_DIS
LIN {X -0.038,Y -351.668,Z 363.622,A 0.000,B 0.000,C 90.000,E1 291.972} C_DIS
LIN {X 0.123,Y -372.240,Z 363.607,A 0.000,B 0.000,C 90.000,E1 289.268} C_DIS
LIN {X -0.068,Y -397.571,Z 363.591,A 0.000,B 0.000,C 90.000,E1 286.441} C_DIS
LIN {X -0.030,Y -415.536,Z 363.581,A 0.000,B 0.000,C 90.000,E1 284.537} C_DIS
LIN {X -0.139,Y -428.370,Z 363.573,A 0.000,B 0.000,C 90.000,E1 283.231} C_DIS
LIN {X 0.110,Y -435.647,Z 363.569,A 0.000,B 0.000,C 90.000,E1 282.411} C_DIS
LIN {X -0.215,Y -442.585,Z 363.565,A 0.000,B 0.000,C 90.000,E1 281.658} C_DIS
LIN {X 0.018,Y -448.945,Z 363.560,A 0.000,B 0.000,C 90.000,E1 280.838} C_DIS
LIN {X 0.039,Y -456.828,Z 363.554,A 0.000,B 0.000,C 90.000,E1 279.792} C_DIS
LIN {X 0.156,Y -464.060,Z 363.549,A 0.000,B 0.000,C 90.000,E1 278.746} C_DIS
LIN {X -0.108,Y -470.582,Z 363.543,A 0.000,B 0.000,C 90.000,E1 277.757} C_DIS
LIN {X 0.105,Y -476.654,Z 363.537,A 0.000,B 0.000,C 90.000,E1 276.720} C_DIS
LIN {X 0.098,Y -480.742,Z 363.533,A 0.000,B 0.000,C 90.000,E1 275.967} C_DIS
LIN {X 0.080,Y -484.237,Z 363.529,A 0.000,B 0.000,C 90.000,E1 275.220} C_DIS
LIN {X 0.092,Y -486.868,Z 363.525,A 0.000,B 0.000,C 90.000,E1 274.473} C_DIS
LIN {X -0.203,Y -488.168,Z 363.522,A 0.000,B 0.000,C 90.000,E1 274.012} C_DIS
LIN {X -0.035,Y -489.097,Z 363.519,A 0.000,B 0.000,C 90.000,E1 273.498} C_DIS
LIN {X 0.170,Y -489.687,Z 363.517,A 0.000,B 0.000,C 90.000,E1 272.980} C_DIS
LIN {X -0.134,Y -489.959,Z 363.514,A 0.000,B 0.000,C 90.000,E1 272.522} C_DIS
LIN {X 0.058,Y -489.971,Z 363.511,A 0.000,B 0.000,C 90.000,E1 272.007} C_DIS
LIN {X -0.222,Y -489.704,Z 363.508,A 0.000,B 0.000,C 90.000,E1 271.547} C_DIS
LIN {X -0.029,Y -489.082,Z 363.506,A 0.000,B 0.000,C 90.000,E1 271.031} C_DIS
LIN {X 0.164,Y -488.136,Z 363.503,A 0.000,B 0.000,C 90.000,E1 270.516} C_DIS
LIN {X -0.134,Y -486.778,Z 363.500,A 0.000,B 0.000,C 90.000,E1 270.057} C_DIS
LIN {X 0.050,Y -484.879,Z 363.497,A 0.000,B 0.000,C 90.000,E1 269.542} C_DIS
LIN {X 0.224,Y -482.414,Z 363.495,A 0.000,B 0.000,C 90.000,E1 269.026} C_DIS
LIN {X -0.101,Y -479.145,Z 363.492,A 0.000,B 0.000,C 90.000,E1 268.568} C_DIS
LIN {X 0.051,Y -474.921,Z 363.489,A 0.000,B 0.000,C 90.000,E1 268.051} C_DIS
LIN {X -0.127,Y -472.350,Z 363.488,A 0.000,B 0.000,C 90.000,E1 267.822} C_DIS
LIN {X 0.216,Y -466.486,Z 363.485,A 0.000,B 0.000,C 90.000,E1 267.306} C_DIS
LIN {X 0.146,Y -459.967,Z 363.483,A 0.000,B 0.000,C 90.000,E1 266.906} C_DIS
LIN {X 0.215,Y -452.902,Z 363.481,A 0.000,B 0.000,C 90.000,E1 266.560} C_DIS
LIN {X -0.097,Y -445.461,Z 363.480,A 0.000,B 0.000,C 90.000,E1 266.331} C_DIS
LIN {X 0.071,Y -437.608,Z 363.478,A 0.000,B 0.000,C 90.000,E1 266.102} C_DIS
LIN {X -0.202,Y -428.711,Z 363.478,A 0.000,B 0.000,C 90.000,E1 265.988} C_DIS
LIN {X -0.069,Y -416.746,Z 363.477,A 0.000,B 0.000,C 90.000,E1 265.869} C_DIS
LIN {X -0.141,Y -413.067,Z 363.477,A 0.000,B 0.000,C 90.000,E1 265.869} C_DIS
LIN {X 0.087,Y -180.915,Z 363.477,A 0.000,B 0.000,C 90.000,E1 265.812} C_DIS
LIN {X 0.083,Y -180.857,Z 363.472,A 0.000,B 0.000,C 90.000,E1 264.951} C_DIS
LIN {X -0.044,Y -178.968,Z 363.444,A 0.000,B 0.000,C 90.000,E1 259.926} C_DIS
LIN {X -0.033,Y -177.923,Z 363.435,A 0.000,B 0.000,C 90.000,E1 258.229} C_DIS
LIN {X -0.018,Y -175.560,Z 363.411,A 0.000,B 0.000,C 90.000,E1 253.976} C_DIS
LIN {X -0.011,Y -172.289,Z 363.387,A 0.000,B 0.000,C 90.000,E1 249.699} C_DIS
LIN {X -0.033,Y -171.768,Z 363.382,A 0.000,B 0.000,C 90.000,E1 248.847} C_DIS
LIN {X -0.041,Y -168.009,Z 363.358,A 0.000,B 0.000,C 90.000,E1 244.537} C_DIS
LIN {X -0.022,Y -166.760,Z 363.349,A 0.000,B 0.000,C 90.000,E1 242.794} C_DIS
LIN {X 0.038,Y -162.740,Z 363.325,A 0.000,B 0.000,C 90.000,E1 238.408} C_DIS
LIN {X 0.099,Y -161.430,Z 363.315,A 0.000,B 0.000,C 90.000,E1 236.628} C_DIS
LIN {X -0.081,Y -157.423,Z 363.290,A 0.000,B 0.000,C 90.000,E1 232.271} C_DIS
LIN {X 0.072,Y -155.426,Z 363.275,A 0.000,B 0.000,C 90.000,E1 229.542} C_DIS
LIN {X 0.002,Y -151.750,Z 363.250,A 0.000,B 0.000,C 90.000,E1 225.081} C_DIS
LIN {X 0.014,Y -149.951,Z 363.235,A 0.000,B 0.000,C 90.000,E1 222.366} C_DIS
LIN {X 0.041,Y -146.794,Z 363.210,A 0.000,B 0.000,C 90.000,E1 217.810} C_DIS
LIN {X -0.058,Y -145.369,Z 363.195,A 0.000,B 0.000,C 90.000,E1 215.105} C_DIS
LIN {X 0.058,Y -142.434,Z 363.164,A 0.000,B 0.000,C 90.000,E1 209.539} C_DIS
LIN {X -0.018,Y -141.424,Z 363.149,A 0.000,B 0.000,C 90.000,E1 206.796} C_DIS
LIN {X -0.037,Y -139.362,Z 363.113,A 0.000,B 0.000,C 90.000,E1 200.301} C_DIS
LIN {X -0.050,Y -138.807,Z 363.097,A 0.000,B 0.000,C 90.000,E1 197.511} C_DIS
LIN {X 0.000,Y -138.350,Z 363.056,A 0.000,B 0.000,C 90.000,E1 190.018} C_DIS
LIN {X -0.024,Y -139.543,Z 363.004,A 0.000,B 0.000,C 90.000,E1 180.688} C_DIS
LIN {X 0.069,Y -141.243,Z 362.973,A 0.000,B 0.000,C 90.000,E1 175.065} C_DIS
LIN {X 0.028,Y -142.612,Z 362.957,A 0.000,B 0.000,C 90.000,E1 172.299} C_DIS
LIN {X -0.019,Y -144.927,Z 362.932,A 0.000,B 0.000,C 90.000,E1 167.701} C_DIS
LIN {X -0.028,Y -147.556,Z 362.911,A 0.000,B 0.000,C 90.000,E1 164.031} C_DIS
LIN {X 0.005,Y -150.160,Z 362.891,A 0.000,B 0.000,C 90.000,E1 160.369} C_DIS
LIN {X 0.014,Y -153.533,Z 362.871,A 0.000,B 0.000,C 90.000,E1 156.741} C_DIS
LIN {X 0.066,Y -156.951,Z 362.851,A 0.000,B 0.000,C 90.000,E1 153.127} C_DIS
LIN {X 0.002,Y -161.056,Z 362.831,A 0.000,B 0.000,C 90.000,E1 149.587} C_DIS
LIN {X 0.087,Y -163.165,Z 362.821,A 0.000,B 0.000,C 90.000,E1 147.788} C_DIS
LIN {X -0.042,Y -167.583,Z 362.802,A 0.000,B 0.000,C 90.000,E1 144.322} C_DIS
LIN {X 0.003,Y -171.413,Z 362.787,A 0.000,B 0.000,C 90.000,E1 141.698} C_DIS
LIN {X 0.043,Y -176.329,Z 362.768,A 0.000,B 0.000,C 90.000,E1 138.243} C_DIS
LIN {X -0.089,Y -180.618,Z 362.754,A 0.000,B 0.000,C 90.000,E1 135.729} C_DIS
LIN {X 0.025,Y -186.019,Z 362.735,A 0.000,B 0.000,C 90.000,E1 132.324} C_DIS
LIN {X -0.058,Y -190.654,Z 362.721,A 0.000,B 0.000,C 90.000,E1 129.850} C_DIS
LIN {X 0.004,Y -196.405,Z 362.703,A 0.000,B 0.000,C 90.000,E1 126.537} C_DIS
LIN {X -0.058,Y -199.585,Z 362.694,A 0.000,B 0.000,C 90.000,E1 124.945} C_DIS
LIN {X 0.123,Y -299.598,Z 362.694,A 0.000,B 0.000,C 90.000,E1 124.898} C_DIS
LIN {X -0.095,Y -303.761,Z 362.693,A 0.000,B 0.000,C 90.000,E1 124.818} C_DIS
LIN {X -0.132,Y -306.972,Z 362.692,A 0.000,B 0.000,C 90.000,E1 124.612} C_DIS
LIN {X -0.063,Y -310.657,Z 362.690,A 0.000,B 0.000,C 90.000,E1 124.199} C_DIS
LIN {X -0.138,Y -312.594,Z 362.688,A 0.000,B 0.000,C 90.000,E1 123.913} C_DIS
LIN {X 0.047,Y -314.122,Z 362.687,A 0.000,B 0.000,C 90.000,E1 123.579} C_DIS
LIN {X -0.102,Y -316.532,Z 362.683,A 0.000,B 0.000,C 90.000,E1 122.959} C_DIS
LIN {X -0.088,Y -327.002,Z 362.667,A 0.000,B 0.000,C 90.000,E1 120.079} C_DIS
LIN {X -0.104,Y -338.841,Z 362.651,A 0.000,B 0.000,C 90.000,E1 117.257} C_DIS
LIN {X 0.066,Y -352.149,Z 362.636,A 0.000,B 0.000,C 90.000,E1 114.463} C_DIS
LIN {X -0.068,Y -365.317,Z 362.623,A 0.000,B 0.000,C 90.000,E1 112.078} C_DIS
LIN {X 0.060,Y -379.841,Z 362.610,A 0.000,B 0.000,C 90.000,E1 109.704} C_DIS
LIN {X 0.081,Y -395.828,Z 362.597,A 0.000,B 0.000,C 90.000,E1 107.402} C_DIS
LIN {X -0.130,Y -413.398,Z 362.584,A 0.000,B 0.000,C 90.000,E1 105.190} C_DIS
LIN {X -0.105,Y -432.647,Z 362.572,A 0.000,B 0.000,C 90.000,E1 103.008} C_DIS
LIN {X 0.084,Y -452.863,Z 362.561,A 0.000,B 0.000,C 90.000,E1 100.950} C_DIS
LIN {X 0.027,Y -473.618,Z 362.551,A 0.000,B 0.000,C 90.000,E1 99.095} C_DIS
LIN {X 0.049,Y -492.059,Z 362.542,A 0.000,B 0.000,C 90.000,E1 97.587} C_DIS
LIN {X -0.149,Y -495.625,Z 362.540,A 0.000,B 0.000,C 90.000,E1 97.182} C_DIS
LIN {X 0.247,Y -496.986,Z 362.538,A 0.000,B 0.000,C 90.000,E1 96.891} C_DIS
LIN {X 0.090,Y -497.991,Z 362.537,A 0.000,B 0.000,C 90.000,E1 96.663} C_DIS
LIN {X -0.138,Y -499.117,Z 362.534,A 0.000,B 0.000,C 90.000,E1 96.201} C_DIS
LIN {X 0.136,Y -499.222,Z 362.532,A 0.000,B 0.000,C 90.000,E1 95.682} C_DIS
LIN {X -0.082,Y -498.322,Z 362.529,A 0.000,B 0.000,C 90.000,E1 95.220} C_DIS
LIN {X 0.194,Y -496.253,Z 362.526,A 0.000,B 0.000,C 90.000,E1 94.702} C_DIS
LIN {X -0.068,Y -492.900,Z 362.524,A 0.000,B 0.000,C 90.000,E1 94.245} C_DIS
LIN {X -0.115,Y -485.420,Z 362.518,A 0.000,B 0.000,C 90.000,E1 93.269} C_DIS
LIN {X 0.190,Y -471.355,Z 362.508,A 0.000,B 0.000,C 90.000,E1 91.489} C_DIS
LIN {X 0.191,Y -450.360,Z 362.493,A 0.000,B 0.000,C 90.000,E1 88.682} C_DIS
LIN {X 0.191,Y -429.653,Z 362.475,A 0.000,B 0.000,C 90.000,E1 85.527} C_DIS
LIN {X 0.155,Y -409.484,Z 362.456,A 0.000,B 0.000,C 90.000,E1 82.008} C_DIS
LIN {X 0.130,Y -396.303,Z 362.442,A 0.000,B 0.000,C 90.000,E1 79.511} C_DIS
LIN {X 0.190,Y -386.069,Z 362.431,A 0.000,B 0.000,C 90.000,E1 77.521} C_DIS
LIN {X 0.140,Y -372.969,Z 362.416,A 0.000,B 0.000,C 90.000,E1 74.936} C_DIS
LIN {X -0.015,Y -362.852,Z 362.405,A 0.000,B 0.000,C 90.000,E1 72.906} C_DIS
LIN {X 0.188,Y -352.764,Z 362.393,A 0.000,B 0.000,C 90.000,E1 70.786} C_DIS
LIN {X -0.130,Y -339.987,Z 362.378,A 0.000,B 0.000,C 90.000,E1 68.103} C_DIS
LIN {X 0.066,Y -324.155,Z 362.357,A 0.000,B 0.000,C 90.000,E1 64.332} C_DIS
LIN {X 0.071,Y -313.358,Z 362.342,A 0.000,B 0.000,C 90.000,E1 61.463} C_DIS
LIN {X 0.127,Y -302.083,Z 362.323,A 0.000,B 0.000,C 90.000,E1 58.201} C_DIS
LIN {X 0.092,Y -291.606,Z 362.305,A 0.000,B 0.000,C 90.000,E1 54.895} C_DIS
LIN {X 0.024,Y -282.079,Z 362.286,A 0.000,B 0.000,C 90.000,E1 51.537} C_DIS
LIN {X 0.146,Y -274.578,Z 362.271,A 0.000,B 0.000,C 90.000,E1 48.771} C_DIS
LIN {X 0.091,Y -268.874,Z 362.260,A 0.000,B 0.000,C 90.000,E1 46.701} C_DIS
LIN {X -0.162,Y -261.288,Z 362.244,A 0.000,B 0.000,C 90.000,E1 43.947} C_DIS
LIN {X 0.088,Y -255.579,Z 362.232,A 0.000,B 0.000,C 90.000,E1 41.757} C_DIS
LIN {X -0.112,Y -249.726,Z 362.220,A 0.000,B 0.000,C 90.000,E1 39.644} C_DIS
LIN {X -0.032,Y -243.785,Z 362.208,A 0.000,B 0.000,C 90.000,E1 37.443} C_DIS
LIN {X -0.006,Y -236.053,Z 362.192,A 0.000,B 0.000,C 90.000,E1 34.485} C_DIS
LIN {X 0.081,Y -228.523,Z 362.175,A 0.000,B 0.000,C 90.000,E1 31.465} C_DIS
LIN {X 0.016,Y -221.452,Z 362.158,A 0.000,B 0.000,C 90.000,E1 28.437} C_DIS
LIN {X -0.070,Y -213.481,Z 362.137,A 0.000,B 0.000,C 90.000,E1 24.591} C_DIS
LIN {X 0.083,Y -207.799,Z 362.119,A 0.000,B 0.000,C 90.000,E1 21.408} C_DIS
LIN {X -0.023,Y -201.707,Z 362.097,A 0.000,B 0.000,C 90.000,E1 17.457} C_DIS
LIN {X -0.056,Y -197.526,Z 362.079,A 0.000,B 0.000,C 90.000,E1 14.245} C_DIS
LIN {X 0.067,Y -193.243,Z 362.056,A 0.000,B 0.000,C 90.000,E1 10.141} C_DIS
LIN {X -0.102,Y -190.118,Z 362.034,A 0.000,B 0.000,C 90.000,E1 6.087} C_DIS
LIN {X -0.034,Y -187.731,Z 361.997,A 0.000,B 0.000,C 90.000,E1 359.542} C_DIS
LIN {X 0.027,Y -189.305,Z 361.942,A 0.000,B 0.000,C 90.000,E1 349.567} C_DIS
LIN {X -0.031,Y -192.171,Z 361.915,A 0.000,B 0.000,C 90.000,E1 344.629} C_DIS
LIN {X 0.073,Y -195.795,Z 361.892,A 0.000,B 0.000,C 90.000,E1 340.496} C_DIS
LIN {X 0.064,Y -200.550,Z 361.869,A 0.000,B 0.000,C 90.000,E1 336.433} C_DIS
LIN {X -0.095,Y -205.113,Z 361.851,A 0.000,B 0.000,C 90.000,E1 333.256} C_DIS
LIN {X -0.018,Y -211.708,Z 361.829,A 0.000,B 0.000,C 90.000,E1 329.253} C_DIS
LIN {X 0.057,Y -218.885,Z 361.807,A 0.000,B 0.000,C 90.000,E1 325.308} C_DIS
LIN {X 0.014,Y -226.990,Z 361.786,A 0.000,B 0.000,C 90.000,E1 321.457} C_DIS
LIN {X 0.051,Y -234.130,Z 361.769,A 0.000,B 0.000,C 90.000,E1 318.405} C_DIS
LIN {X -0.131,Y -243.243,Z 361.750,A 0.000,B 0.000,C 90.000,E1 315.081} C_DIS
LIN {X -0.041,Y -252.337,Z 361.734,A 0.000,B 0.000,C 90.000,E1 312.123} C_DIS
LIN {X 0.116,Y -261.003,Z 361.720,A 0.000,B 0.000,C 90.000,E1 309.564} C_DIS
LIN {X -0.082,Y -272.831,Z 361.702,A 0.000,B 0.000,C 90.000,E1 306.423} C_DIS
LIN {X 0.053,Y -284.189,Z 361.687,A 0.000,B 0.000,C 90.000,E1 303.627} C_DIS
LIN {X 0.013,Y -298.287,Z 361.670,A 0.000,B 0.000,C 90.000,E1 300.590} C_DIS
LIN {X -0.113,Y -312.250,Z 361.655,A 0.000,B 0.000,C 90.000,E1 297.975} C_DIS
LIN {X -0.120,Y -321.846,Z 361.646,A 0.000,B 0.000,C 90.000,E1 296.360} C_DIS
LIN {X -0.076,Y -338.583,Z 361.632,A 0.000,B 0.000,C 90.000,E1 293.823} C_DIS
LIN {X -0.042,Y -354.163,Z 361.620,A 0.000,B 0.000,C 90.000,E1 291.663} C_DIS
LIN {X -0.117,Y -370.305,Z 361.609,A 0.000,B 0.000,C 90.000,E1 289.577} C_DIS
LIN {X -0.001,Y -395.572,Z 361.593,A 0.000,B 0.000,C 90.000,E1 286.677} C_DIS
LIN {X 0.005,Y -413.466,Z 361.582,A 0.000,B 0.000,C 90.000,E1 284.773} C_DIS
LIN {X 0.094,Y -428.795,Z 361.573,A 0.000,B 0.000,C 90.000,E1 283.175} C_DIS
LIN {X -0.123,Y -436.047,Z 361.569,A 0.000,B 0.000,C 90.000,E1 282.411} C_DIS
LIN {X 0.041,Y -442.932,Z 361.564,A 0.000,B 0.000,C 90.000,E1 281.591} C_DIS
LIN {X 0.192,Y -449.242,Z 361.560,A 0.000,B 0.000,C 90.000,E1 280.782} C_DIS
LIN {X -0.151,Y -457.063,Z 361.554,A 0.000,B 0.000,C 90.000,E1 279.782} C_DIS
LIN {X -0.113,Y -464.248,Z 361.549,A 0.000,B 0.000,C 90.000,E1 278.746} C_DIS
LIN {X 0.088,Y -470.733,Z 361.543,A 0.000,B 0.000,C 90.000,E1 277.701} C_DIS
LIN {X -0.168,Y -476.782,Z 361.537,A 0.000,B 0.000,C 90.000,E1 276.720} C_DIS
LIN {X -0.175,Y -480.832,Z 361.533,A 0.000,B 0.000,C 90.000,E1 275.967} C_DIS
LIN {X -0.194,Y -484.242,Z 361.529,A 0.000,B 0.000,C 90.000,E1 275.220} C_DIS
LIN {X 0.114,Y -485.250,Z 361.527,A 0.000,B 0.000,C 90.000,E1 274.935} C_DIS
LIN {X -0.184,Y -486.860,Z 361.525,A 0.000,B 0.000,C 90.000,E1 274.473} C_DIS
LIN {X 0.007,Y -488.128,Z 361.522,A 0.000,B 0.000,C 90.000,E1 273.955} C_DIS
LIN {X 0.175,Y -488.991,Z 361.519,A 0.000,B 0.000,C 90.000,E1 273.440} C_DIS
LIN {X -0.108,Y -489.545,Z 361.516,A 0.000,B 0.000,C 90.000,E1 272.980} C_DIS
LIN {X 0.077,Y -489.775,Z 361.514,A 0.000,B 0.000,C 90.000,E1 272.465} C_DIS
LIN {X -0.221,Y -489.731,Z 361.511,A 0.000,B 0.000,C 90.000,E1 272.007} C_DIS
LIN {X -0.013,Y -489.414,Z 361.508,A 0.000,B 0.000,C 90.000,E1 271.489} C_DIS
LIN {X 0.178,Y -488.774,Z 361.506,A 0.000,B 0.000,C 90.000,E1 270.974} C_DIS
LIN {X -0.119,Y -487.788,Z 361.503,A 0.000,B 0.000,C 90.000,E1 270.516} C_DIS
LIN {X 0.069,Y -486.386,Z 361.500,A 0.000,B 0.000,C 90.000,E1 270.000} C_DIS
LIN {X -0.234,Y -484.465,Z 361.497,A 0.000,B 0.000,C 90.000,E1 269.542} C_DIS
LIN {X -0.061,Y -481.977,Z 361.495,A 0.000,B 0.000,C 90.000,E1 269.026} C_DIS
LIN {X -0.224,Y -480.467,Z 361.493,A 0.000,B 0.000,C 90.000,E1 268.797} C_DIS
LIN {X -0.080,Y -476.684,Z 361.490,A 0.000,B 0.000,C 90.000,E1 268.282} C_DIS
LIN {X 0.240,Y -474.447,Z 361.489,A 0.000,B 0.000,C 90.000,E1 267.993} C_DIS
LIN {X -0.119,Y -468.903,Z 361.486,A 0.000,B 0.000,C 90.000,E1 267.535} C_DIS
LIN {X -0.082,Y -465.947,Z 361.485,A 0.000,B 0.000,C 90.000,E1 267.306} C_DIS
LIN {X -0.149,Y -459.442,Z 361.483,A 0.000,B 0.000,C 90.000,E1 266.906} C_DIS
LIN {X -0.041,Y -452.383,Z 361.481,A 0.000,B 0.000,C 90.000,E1 266.560} C_DIS
LIN {X 0.117,Y -444.877,Z 361.479,A 0.000,B 0.000,C 90.000,E1 266.274} C_DIS
LIN {X -0.140,Y -436.898,Z 361.478,A 0.000,B 0.000,C 90.000,E1 266.102} C_DIS
LIN {X 0.094,Y -427.858,Z 361.477,A 0.000,B 0.000,C 90.000,E1 265.927} C_DIS
LIN {X -0.044,Y -419.457,Z 361.477,A 0.000,B 0.000,C 90.000,E1 265.869} C_DIS
LIN {X -0.180,Y -414.794,Z 361.477,A 0.000,B 0.000,C 90.000,E1 265.869} C_DIS
LIN {X 0.072,Y -180.914,Z 361.477,A 0.000,B 0.000,C 90.000,E1 265.812} C_DIS
LIN {X 0.044,Y -180.803,Z 361.471,A 0.000,B 0.000,C 90.000,E1 264.780} C_DIS
LIN {X -0.033,Y -178.824,Z 361.442,A 0.000,B 0.000,C 90.000,E1 259.567} C_DIS
LIN {X 0.049,Y -175.870,Z 361.414,A 0.000,B 0.000,C 90.000,E1 254.448} C_DIS
LIN {X 0.043,Y -173.840,Z 361.399,A 0.000,B 0.000,C 90.000,E1 251.891} C_DIS
LIN {X 0.033,Y -171.508,Z 361.380,A 0.000,B 0.000,C 90.000,E1 248.465} C_DIS
LIN {X 0.019,Y -167.735,Z 361.356,A 0.000,B 0.000,C 90.000,E1 244.152} C_DIS
LIN {X 0.035,Y -166.433,Z 361.347,A 0.000,B 0.000,C 90.000,E1 242.410} C_DIS
LIN {X -0.051,Y -163.153,Z 361.327,A 0.000,B 0.000,C 90.000,E1 238.948} C_DIS
LIN {X -0.002,Y -161.108,Z 361.313,A 0.000,B 0.000,C 90.000,E1 236.294} C_DIS
LIN {X -0.018,Y -157.835,Z 361.293,A 0.000,B 0.000,C 90.000,E1 232.763} C_DIS
LIN {X 0.045,Y -155.868,Z 361.278,A 0.000,B 0.000,C 90.000,E1 230.070} C_DIS
LIN {X -0.007,Y -152.118,Z 361.253,A 0.000,B 0.000,C 90.000,E1 225.607} C_DIS
LIN {X 0.007,Y -150.368,Z 361.238,A 0.000,B 0.000,C 90.000,E1 222.894} C_DIS
LIN {X -0.070,Y -147.102,Z 361.213,A 0.000,B 0.000,C 90.000,E1 218.382} C_DIS
LIN {X 0.040,Y -145.671,Z 361.198,A 0.000,B 0.000,C 90.000,E1 215.598} C_DIS
LIN {X 0.043,Y -143.053,Z 361.172,A 0.000,B 0.000,C 90.000,E1 211.003} C_DIS
LIN {X -0.022,Y -141.676,Z 361.152,A 0.000,B 0.000,C 90.000,E1 207.334} C_DIS
LIN {X -0.043,Y -139.455,Z 361.116,A 0.000,B 0.000,C 90.000,E1 200.844} C_DIS
LIN {X 0.007,Y -139.188,Z 361.105,A 0.000,B 0.000,C 90.000,E1 198.960} C_DIS
LIN {X 0.031,Y -138.322,Z 361.053,A 0.000,B 0.000,C 90.000,E1 189.613} C_DIS
LIN {X 0.038,Y -139.458,Z 361.007,A 0.000,B 0.000,C 90.000,E1 181.203} C_DIS
LIN {X -0.021,Y -141.011,Z 360.976,A 0.000,B 0.000,C 90.000,E1 175.641} C_DIS
LIN {X 0.069,Y -142.765,Z 360.955,A 0.000,B 0.000,C 90.000,E1 171.894} C_DIS
LIN {X 0.025,Y -145.172,Z 360.929,A 0.000,B 0.000,C 90.000,E1 167.297} C_DIS
LIN {X 0.058,Y -147.795,Z 360.909,A 0.000,B 0.000,C 90.000,E1 163.614} C_DIS
LIN {X -0.047,Y -150.478,Z 360.889,A 0.000,B 0.000,C 90.000,E1 160.007} C_DIS
LIN {X 0.027,Y -153.931,Z 360.869,A 0.000,B 0.000,C 90.000,E1 156.357} C_DIS
LIN {X -0.049,Y -157.342,Z 360.849,A 0.000,B 0.000,C 90.000,E1 152.794} C_DIS
LIN {X 0.034,Y -161.536,Z 360.829,A 0.000,B 0.000,C 90.000,E1 149.203} C_DIS
LIN {X 0.047,Y -165.735,Z 360.809,A 0.000,B 0.000,C 90.000,E1 145.674} C_DIS
LIN {X 0.035,Y -170.686,Z 360.790,A 0.000,B 0.000,C 90.000,E1 142.190} C_DIS
LIN {X -0.053,Y -175.559,Z 360.771,A 0.000,B 0.000,C 90.000,E1 138.771} C_DIS
LIN {X 0.067,Y -181.178,Z 360.752,A 0.000,B 0.000,C 90.000,E1 135.324} C_DIS
LIN {X -0.065,Y -186.636,Z 360.733,A 0.000,B 0.000,C 90.000,E1 132.000} C_DIS
LIN {X 0.005,Y -191.243,Z 360.719,A 0.000,B 0.000,C 90.000,E1 129.483} C_DIS
LIN {X -0.073,Y -197.061,Z 360.701,A 0.000,B 0.000,C 90.000,E1 126.217} C_DIS
LIN {X -0.059,Y -199.682,Z 360.694,A 0.000,B 0.000,C 90.000,E1 124.898} C_DIS
LIN {X -0.141,Y -299.410,Z 360.694,A 0.000,B 0.000,C 90.000,E1 124.898} C_DIS
LIN {X 0.116,Y -301.410,Z 360.694,A 0.000,B 0.000,C 90.000,E1 124.818} C_DIS
LIN {X 0.015,Y -306.734,Z 360.692,A 0.000,B 0.000,C 90.000,E1 124.565} C_DIS
LIN {X 0.026,Y -309.916,Z 360.690,A 0.000,B 0.000,C 90.000,E1 124.246} C_DIS
LIN {X -0.089,Y -313.536,Z 360.687,A 0.000,B 0.000,C 90.000,E1 123.706} C_DIS
LIN {X -0.041,Y -315.009,Z 360.685,A 0.000,B 0.000,C 90.000,E1 123.372} C_DIS
LIN {X -0.166,Y -327.844,Z 360.666,A 0.000,B 0.000,C 90.000,E1 119.873} C_DIS
LIN {X 0.140,Y -339.788,Z 360.650,A 0.000,B 0.000,C 90.000,E1 117.001} C_DIS
LIN {X 0.022,Y -353.219,Z 360.635,A 0.000,B 0.000,C 90.000,E1 114.259} C_DIS
LIN {X 0.105,Y -366.501,Z 360.621,A 0.000,B 0.000,C 90.000,E1 111.844} C_DIS
LIN {X 0.048,Y -381.147,Z 360.608,A 0.000,B 0.000,C 90.000,E1 109.504} C_DIS
LIN {X -0.032,Y -397.268,Z 360.596,A 0.000,B 0.000,C 90.000,E1 107.221} C_DIS
LIN {X 0.186,Y -414.980,Z 360.583,A 0.000,B 0.000,C 90.000,E1 104.954} C_DIS
LIN {X -0.142,Y -434.363,Z 360.571,A 0.000,B 0.000,C 90.000,E1 102.827} C_DIS
LIN {X 0.078,Y -454.629,Z 360.560,A 0.000,B 0.000,C 90.000,E1 100.782} C_DIS
LIN {X 0.219,Y -475.428,Z 360.550,A 0.000,B 0.000,C 90.000,E1 98.916} C_DIS
LIN {X 0.103,Y -491.326,Z 360.543,A 0.000,B 0.000,C 90.000,E1 97.644} C_DIS
LIN {X 0.000,Y -495.204,Z 360.540,A 0.000,B 0.000,C 90.000,E1 97.239} C_DIS
LIN {X -0.100,Y -496.722,Z 360.539,A 0.000,B 0.000,C 90.000,E1 97.004} C_DIS
LIN {X 0.234,Y -497.853,Z 360.537,A 0.000,B 0.000,C 90.000,E1 96.720} C_DIS
LIN {X 0.005,Y -499.183,Z 360.535,A 0.000,B 0.000,C 90.000,E1 96.258} C_DIS
LIN {X -0.219,Y -499.469,Z 360.532,A 0.000,B 0.000,C 90.000,E1 95.796} C_DIS
LIN {X 0.060,Y -498.758,Z 360.529,A 0.000,B 0.000,C 90.000,E1 95.277} C_DIS
LIN {X -0.200,Y -496.927,Z 360.527,A 0.000,B 0.000,C 90.000,E1 94.821} C_DIS
LIN {X 0.205,Y -495.479,Z 360.525,A 0.000,B 0.000,C 90.000,E1 94.531} C_DIS
LIN {X 0.179,Y -488.262,Z 360.520,A 0.000,B 0.000,C 90.000,E1 93.555} C_DIS
LIN {X 0.074,Y -480.350,Z 360.514,A 0.000,B 0.000,C 90.000,E1 92.579} C_DIS
LIN {X -0.076,Y -454.892,Z 360.496,A 0.000,B 0.000,C 90.000,E1 89.312} C_DIS
LIN {X 0.177,Y -437.132,Z 360.482,A 0.000,B 0.000,C 90.000,E1 86.674} C_DIS
LIN {X -0.054,Y -420.831,Z 360.467,A 0.000,B 0.000,C 90.000,E1 84.033} C_DIS
LIN {X -0.139,Y -405.767,Z 360.452,A 0.000,B 0.000,C 90.000,E1 81.310} C_DIS
LIN {X -0.018,Y -395.543,Z 360.441,A 0.000,B 0.000,C 90.000,E1 79.342} C_DIS
LIN {X 0.028,Y -385.326,Z 360.430,A 0.000,B 0.000,C 90.000,E1 77.353} C_DIS
LIN {X 0.043,Y -373.689,Z 360.417,A 0.000,B 0.000,C 90.000,E1 75.046} C_DIS
LIN {X -0.118,Y -362.107,Z 360.404,A 0.000,B 0.000,C 90.000,E1 72.725} C_DIS
LIN {X 0.069,Y -352.007,Z 360.392,A 0.000,B 0.000,C 90.000,E1 70.604} C_DIS
LIN {X 0.178,Y -339.237,Z 360.377,A 0.000,B 0.000,C 90.000,E1 67.847} C_DIS
LIN {X -0.052,Y -324.722,Z 360.358,A 0.000,B 0.000,C 90.000,E1 64.460} C_DIS
LIN {X -0.027,Y -313.905,Z 360.342,A 0.000,B 0.000,C 90.000,E1 61.591} C_DIS
LIN {X 0.079,Y -301.509,Z 360.322,A 0.000,B 0.000,C 90.000,E1 57.995} C_DIS
LIN {X 0.026,Y -290.124,Z 360.302,A 0.000,B 0.000,C 90.000,E1 54.356} C_DIS
LIN {X -0.006,Y -282.536,Z 360.287,A 0.000,B 0.000,C 90.000,E1 51.662} C_DIS
LIN {X -0.046,Y -275.025,Z 360.272,A 0.000,B 0.000,C 90.000,E1 48.933} C_DIS
LIN {X 0.096,Y -269.327,Z 360.260,A 0.000,B 0.000,C 90.000,E1 46.824} C_DIS
LIN {X 0.043,Y -261.746,Z 360.245,A 0.000,B 0.000,C 90.000,E1 44.028} C_DIS
LIN {X -0.065,Y -256.055,Z 360.233,A 0.000,B 0.000,C 90.000,E1 41.919} C_DIS
LIN {X 0.103,Y -250.245,Z 360.221,A 0.000,B 0.000,C 90.000,E1 39.725} C_DIS
LIN {X -0.006,Y -244.313,Z 360.209,A 0.000,B 0.000,C 90.000,E1 37.569} C_DIS
LIN {X 0.028,Y -236.540,Z 360.192,A 0.000,B 0.000,C 90.000,E1 34.612} C_DIS
LIN {X 0.124,Y -228.980,Z 360.176,A 0.000,B 0.000,C 90.000,E1 31.592} C_DIS
LIN {X 0.065,Y -221.862,Z 360.159,A 0.000,B 0.000,C 90.000,E1 28.565} C_DIS
LIN {X -0.010,Y -213.853,Z 360.137,A 0.000,B 0.000,C 90.000,E1 24.719} C_DIS
LIN {X -0.042,Y -208.124,Z 360.120,A 0.000,B 0.000,C 90.000,E1 21.589} C_DIS
LIN {X -0.062,Y -203.146,Z 360.102,A 0.000,B 0.000,C 90.000,E1 18.417} C_DIS
LIN {X -0.007,Y -198.729,Z 360.084,A 0.000,B 0.000,C 90.000,E1 15.190} C_DIS
LIN {X 0.002,Y -194.228,Z 360.062,A 0.000,B 0.000,C 90.000,E1 11.130} C_DIS
LIN {X 0.076,Y -190.778,Z 360.039,A 0.000,B 0.000,C 90.000,E1 7.011} C_DIS
LIN {X -0.025,Y -188.096,Z 360.007,A 0.000,B 0.000,C 90.000,E1 1.260} C_DIS
LIN {X 0.051,Y -188.140,Z 359.961,A 0.000,B 0.000,C 90.000,E1 352.875} C_DIS
LIN {X -0.076,Y -190.490,Z 359.928,A 0.000,B 0.000,C 90.000,E1 347.117} C_DIS
LIN {X -0.089,Y -194.210,Z 359.901,A 0.000,B 0.000,C 90.000,E1 342.181} C_DIS
LIN {X -0.106,Y -198.486,Z 359.878,A 0.000,B 0.000,C 90.000,E1 338.103} C_DIS
LIN {X 0.022,Y -203.851,Z 359.856,A 0.000,B 0.000,C 90.000,E1 334.024} C_DIS
LIN {X -0.049,Y -208.891,Z 359.838,A 0.000,B 0.000,C 90.000,E1 330.845} C_DIS
LIN {X 0.029,Y -214.432,Z 359.820,A 0.000,B 0.000,C 90.000,E1 327.661} C_DIS
LIN {X -0.074,Y -220.351,Z 359.803,A 0.000,B 0.000,C 90.000,E1 324.562} C_DIS
LIN {X 0.001,Y -226.912,Z 359.786,A 0.000,B 0.000,C 90.000,E1 321.457} C_DIS
LIN {X 0.035,Y -234.072,Z 359.769,A 0.000,B 0.000,C 90.000,E1 318.405} C_DIS
LIN {X 0.023,Y -243.183,Z 359.750,A 0.000,B 0.000,C 90.000,E1 315.040} C_DIS
LIN {X -0.061,Y -252.297,Z 359.734,A 0.000,B 0.000,C 90.000,E1 312.123} C_DIS
LIN {X 0.094,Y -260.953,Z 359.720,A 0.000,B 0.000,C 90.000,E1 309.564} C_DIS
LIN {X 0.113,Y -272.772,Z 359.702,A 0.000,B 0.000,C 90.000,E1 306.377} C_DIS
LIN {X 0.025,Y -284.197,Z 359.687,A 0.000,B 0.000,C 90.000,E1 303.627} C_DIS
LIN {X -0.010,Y -296.726,Z 359.672,A 0.000,B 0.000,C 90.000,E1 300.924} C_DIS
LIN {X -0.029,Y -310.539,Z 359.657,A 0.000,B 0.000,C 90.000,E1 298.281} C_DIS
LIN {X -0.072,Y -320.032,Z 359.648,A 0.000,B 0.000,C 90.000,E1 296.668} C_DIS
LIN {X -0.096,Y -338.808,Z 359.632,A 0.000,B 0.000,C 90.000,E1 293.823} C_DIS
LIN {X -0.083,Y -352.159,Z 359.622,A 0.000,B 0.000,C 90.000,E1 291.972} C_DIS
LIN {X -0.127,Y -370.608,Z 359.609,A 0.000,B 0.000,C 90.000,E1 289.577} C_DIS
LIN {X 0.042,Y -395.795,Z 359.593,A 0.000,B 0.000,C 90.000,E1 286.677} C_DIS
LIN {X 0.126,Y -413.568,Z 359.582,A 0.000,B 0.000,C 90.000,E1 284.773} C_DIS
LIN {X -0.099,Y -428.649,Z 359.573,A 0.000,B 0.000,C 90.000,E1 283.231} C_DIS
LIN {X 0.055,Y -435.950,Z 359.569,A 0.000,B 0.000,C 90.000,E1 282.411} C_DIS
LIN {X 0.220,Y -442.794,Z 359.565,A 0.000,B 0.000,C 90.000,E1 281.591} C_DIS
LIN {X -0.069,Y -449.107,Z 359.560,A 0.000,B 0.000,C 90.000,E1 280.838} C_DIS
LIN {X -0.047,Y -456.885,Z 359.554,A 0.000,B 0.000,C 90.000,E1 279.792} C_DIS
LIN {X 0.070,Y -464.062,Z 359.549,A 0.000,B 0.000,C 90.000,E1 278.746} C_DIS
LIN {X 0.050,Y -472.101,Z 359.542,A 0.000,B 0.000,C 90.000,E1 277.473} C_DIS
LIN {X -0.133,Y -477.973,Z 359.536,A 0.000,B 0.000,C 90.000,E1 276.486} C_DIS
LIN {X -0.178,Y -481.813,Z 359.532,A 0.000,B 0.000,C 90.000,E1 275.739} C_DIS
LIN {X 0.119,Y -483.007,Z 359.530,A 0.000,B 0.000,C 90.000,E1 275.454} C_DIS
LIN {X -0.188,Y -485.033,Z 359.528,A 0.000,B 0.000,C 90.000,E1 274.992} C_DIS
LIN {X -0.009,Y -486.672,Z 359.525,A 0.000,B 0.000,C 90.000,E1 274.473} C_DIS
LIN {X 0.182,Y -487.952,Z 359.522,A 0.000,B 0.000,C 90.000,E1 273.955} C_DIS
LIN {X -0.139,Y -488.824,Z 359.519,A 0.000,B 0.000,C 90.000,E1 273.498} C_DIS
LIN {X 0.066,Y -489.336,Z 359.517,A 0.000,B 0.000,C 90.000,E1 272.980} C_DIS
LIN {X -0.240,Y -489.575,Z 359.514,A 0.000,B 0.000,C 90.000,E1 272.522} C_DIS
LIN {X -0.050,Y -489.497,Z 359.511,A 0.000,B 0.000,C 90.000,E1 272.007} C_DIS
LIN {X 0.156,Y -489.178,Z 359.508,A 0.000,B 0.000,C 90.000,E1 271.489} C_DIS
LIN {X -0.143,Y -488.552,Z 359.506,A 0.000,B 0.000,C 90.000,E1 271.031} C_DIS
LIN {X 0.048,Y -487.551,Z 359.503,A 0.000,B 0.000,C 90.000,E1 270.516} C_DIS
LIN {X 0.234,Y -486.176,Z 359.500,A 0.000,B 0.000,C 90.000,E1 270.000} C_DIS
LIN {X -0.227,Y -483.186,Z 359.496,A 0.000,B 0.000,C 90.000,E1 269.312} C_DIS
LIN {X -0.065,Y -480.361,Z 359.493,A 0.000,B 0.000,C 90.000,E1 268.797} C_DIS
LIN {X 0.078,Y -476.663,Z 359.491,A 0.000,B 0.000,C 90.000,E1 268.282} C_DIS
LIN {X -0.077,Y -474.463,Z 359.489,A 0.000,B 0.000,C 90.000,E1 268.051} C_DIS
LIN {X 0.216,Y -471.924,Z 359.488,A 0.000,B 0.000,C 90.000,E1 267.764} C_DIS
LIN {X 0.036,Y -469.069,Z 359.486,A 0.000,B 0.000,C 90.000,E1 267.535} C_DIS
LIN {X 0.043,Y -466.122,Z 359.485,A 0.000,B 0.000,C 90.000,E1 267.306} C_DIS
LIN {X 0.050,Y -462.784,Z 359.484,A 0.000,B 0.000,C 90.000,E1 267.078} C_DIS
LIN {X -0.108,Y -459.586,Z 359.483,A 0.000,B 0.000,C 90.000,E1 266.906} C_DIS
LIN {X 0.217,Y -455.909,Z 359.482,A 0.000,B 0.000,C 90.000,E1 266.674} C_DIS
LIN {X 0.048,Y -448.415,Z 359.480,A 0.000,B 0.000,C 90.000,E1 266.388} C_DIS
LIN {X 0.015,Y -440.683,Z 359.479,A 0.000,B 0.000,C 90.000,E1 266.159} C_DIS
LIN {X -0.002,Y -432.040,Z 359.478,A 0.000,B 0.000,C 90.000,E1 265.988} C_DIS
LIN {X 0.032,Y -422.276,Z 359.477,A 0.000,B 0.000,C 90.000,E1 265.869} C_DIS
LIN {X -0.176,Y -416.984,Z 359.477,A 0.000,B 0.000,C 90.000,E1 265.869} C_DIS
LIN {X 0.074,Y -180.915,Z 359.477,A 0.000,B 0.000,C 90.000,E1 265.812} C_DIS
LIN {X 0.014,Y -180.851,Z 359.472,A 0.000,B 0.000,C 90.000,E1 264.951} C_DIS
LIN {X 0.096,Y -178.961,Z 359.444,A 0.000,B 0.000,C 90.000,E1 259.859} C_DIS
LIN {X -0.012,Y -177.369,Z 359.430,A 0.000,B 0.000,C 90.000,E1 257.353} C_DIS
LIN {X 0.082,Y -175.542,Z 359.411,A 0.000,B 0.000,C 90.000,E1 253.921} C_DIS
LIN {X -0.078,Y -172.276,Z 359.387,A 0.000,B 0.000,C 90.000,E1 249.699} C_DIS
LIN {X -0.037,Y -171.754,Z 359.382,A 0.000,B 0.000,C 90.000,E1 248.827} C_DIS
LIN {X -0.021,Y -167.353,Z 359.354,A 0.000,B 0.000,C 90.000,E1 243.640} C_DIS
LIN {X 0.061,Y -166.742,Z 359.349,A 0.000,B 0.000,C 90.000,E1 242.743} C_DIS
LIN {X -0.027,Y -162.721,Z 359.324,A 0.000,B 0.000,C 90.000,E1 238.408} C_DIS
LIN {X 0.035,Y -161.412,Z 359.315,A 0.000,B 0.000,C 90.000,E1 236.628} C_DIS
LIN {X 0.077,Y -157.405,Z 359.290,A 0.000,B 0.000,C 90.000,E1 232.190} C_DIS
LIN {X 0.009,Y -155.405,Z 359.275,A 0.000,B 0.000,C 90.000,E1 229.542} C_DIS
LIN {X -0.060,Y -151.735,Z 359.250,A 0.000,B 0.000,C 90.000,E1 225.081} C_DIS
LIN {X -0.048,Y -149.931,Z 359.235,A 0.000,B 0.000,C 90.000,E1 222.366} C_DIS
LIN {X -0.019,Y -146.780,Z 359.210,A 0.000,B 0.000,C 90.000,E1 217.810} C_DIS
LIN {X 0.084,Y -145.352,Z 359.195,A 0.000,B 0.000,C 90.000,E1 215.025} C_DIS
LIN {X -0.001,Y -142.424,Z 359.164,A 0.000,B 0.000,C 90.000,E1 209.539} C_DIS
LIN {X 0.048,Y -141.412,Z 359.149,A 0.000,B 0.000,C 90.000,E1 206.744} C_DIS
LIN {X 0.035,Y -139.359,Z 359.113,A 0.000,B 0.000,C 90.000,E1 200.248} C_DIS
LIN {X 0.023,Y -138.801,Z 359.097,A 0.000,B 0.000,C 90.000,E1 197.457} C_DIS
LIN {X -0.059,Y -138.349,Z 359.056,A 0.000,B 0.000,C 90.000,E1 190.018} C_DIS
LIN {X -0.043,Y -139.366,Z 359.009,A 0.000,B 0.000,C 90.000,E1 181.604} C_DIS
LIN {X 0.009,Y -141.254,Z 358.973,A 0.000,B 0.000,C 90.000,E1 175.065} C_DIS
LIN {X -0.032,Y -142.622,Z 358.957,A 0.000,B 0.000,C 90.000,E1 172.299} C_DIS
LIN {X 0.061,Y -144.942,Z 358.931,A 0.000,B 0.000,C 90.000,E1 167.645} C_DIS
LIN {X 0.054,Y -147.570,Z 358.911,A 0.000,B 0.000,C 90.000,E1 163.976} C_DIS
LIN {X -0.057,Y -150.180,Z 358.891,A 0.000,B 0.000,C 90.000,E1 160.369} C_DIS
LIN {X -0.050,Y -153.557,Z 358.871,A 0.000,B 0.000,C 90.000,E1 156.741} C_DIS
LIN {X 0.002,Y -156.975,Z 358.851,A 0.000,B 0.000,C 90.000,E1 153.127} C_DIS
LIN {X 0.076,Y -161.086,Z 358.831,A 0.000,B 0.000,C 90.000,E1 149.537} C_DIS
LIN {X 0.021,Y -163.191,Z 358.821,A 0.000,B 0.000,C 90.000,E1 147.788} C_DIS
LIN {X 0.028,Y -167.615,Z 358.802,A 0.000,B 0.000,C 90.000,E1 144.276} C_DIS
LIN {X -0.064,Y -171.442,Z 358.787,A 0.000,B 0.000,C 90.000,E1 141.698} C_DIS
LIN {X -0.026,Y -176.363,Z 358.768,A 0.000,B 0.000,C 90.000,E1 138.243} C_DIS
LIN {X 0.096,Y -180.655,Z 358.754,A 0.000,B 0.000,C 90.000,E1 135.648} C_DIS
LIN {X 0.080,Y -186.057,Z 358.735,A 0.000,B 0.000,C 90.000,E1 132.285} C_DIS
LIN {X 0.017,Y -190.694,Z 358.721,A 0.000,B 0.000,C 90.000,E1 129.806} C_DIS
LIN {X 0.049,Y -196.446,Z 358.703,A 0.000,B 0.000,C 90.000,E1 126.503} C_DIS
LIN {X 0.037,Y -199.790,Z 358.693,A 0.000,B 0.000,C 90.000,E1 124.818} C_DIS
LIN {X 0.001,Y -299.924,Z 358.693,A 0.000,B 0.000,C 90.000,E1 124.818} C_DIS
LIN {X 0.113,Y -305.238,Z 358.692,A 0.000,B 0.000,C 90.000,E1 124.612} C_DIS
LIN {X -0.028,Y -307.712,Z 358.691,A 0.000,B 0.000,C 90.000,E1 124.452} C_DIS
LIN {X 0.024,Y -311.028,Z 358.689,A 0.000,B 0.000,C 90.000,E1 124.072} C_DIS
LIN {X -0.086,Y -312.988,Z 358.688,A 0.000,B 0.000,C 90.000,E1 123.785} C_DIS
LIN {X 0.064,Y -314.526,Z 358.686,A 0.000,B 0.000,C 90.000,E1 123.452} C_DIS
LIN {X -0.084,Y -316.911,Z 358.682,A 0.000,B 0.000,C 90.000,E1 122.832} C_DIS
LIN {X 0.110,Y -327.436,Z 358.666,A 0.000,B 0.000,C 90.000,E1 119.922} C_DIS
LIN {X -0.054,Y -339.335,Z 358.651,A 0.000,B 0.000,C 90.000,E1 117.129} C_DIS
LIN {X 0.132,Y -352.709,Z 358.635,A 0.000,B 0.000,C 90.000,E1 114.335} C_DIS
LIN {X -0.125,Y -365.939,Z 358.622,A 0.000,B 0.000,C 90.000,E1 111.972} C_DIS
LIN {X 0.157,Y -380.531,Z 358.609,A 0.000,B 0.000,C 90.000,E1 109.577} C_DIS
LIN {X 0.195,Y -396.591,Z 358.596,A 0.000,B 0.000,C 90.000,E1 107.275} C_DIS
LIN {X 0.001,Y -414.240,Z 358.584,A 0.000,B 0.000,C 90.000,E1 105.064} C_DIS
LIN {X 0.054,Y -433.562,Z 358.572,A 0.000,B 0.000,C 90.000,E1 102.883} C_DIS
LIN {X -0.223,Y -453.806,Z 358.560,A 0.000,B 0.000,C 90.000,E1 100.894} C_DIS
LIN {X -0.152,Y -474.586,Z 358.550,A 0.000,B 0.000,C 90.000,E1 99.029} C_DIS
LIN {X 0.165,Y -490.481,Z 358.543,A 0.000,B 0.000,C 90.000,E1 97.701} C_DIS
LIN {X -0.161,Y -492.930,Z 358.542,A 0.000,B 0.000,C 90.000,E1 97.530} C_DIS
LIN {X 0.032,Y -496.369,Z 358.539,A 0.000,B 0.000,C 90.000,E1 97.068} C_DIS
LIN {X -0.062,Y -497.639,Z 358.538,A 0.000,B 0.000,C 90.000,E1 96.834} C_DIS
LIN {X -0.216,Y -498.567,Z 358.537,A 0.000,B 0.000,C 90.000,E1 96.606} C_DIS
LIN {X 0.055,Y -499.565,Z 358.534,A 0.000,B 0.000,C 90.000,E1 96.087} C_DIS
LIN {X -0.164,Y -499.552,Z 358.531,A 0.000,B 0.000,C 90.000,E1 95.625} C_DIS
LIN {X 0.117,Y -498.524,Z 358.528,A 0.000,B 0.000,C 90.000,E1 95.106} C_DIS
LIN {X -0.011,Y -497.580,Z 358.527,A 0.000,B 0.000,C 90.000,E1 94.878} C_DIS
LIN {X -0.099,Y -496.291,Z 358.526,A 0.000,B 0.000,C 90.000,E1 94.645} C_DIS
LIN {X 0.024,Y -491.042,Z 358.522,A 0.000,B 0.000,C 90.000,E1 93.898} C_DIS
LIN {X -0.050,Y -483.348,Z 358.516,A 0.000,B 0.000,C 90.000,E1 92.922} C_DIS
LIN {X 0.071,Y -463.405,Z 358.502,A 0.000,B 0.000,C 90.000,E1 90.401} C_DIS
LIN {X 0.099,Y -444.872,Z 358.488,A 0.000,B 0.000,C 90.000,E1 87.822} C_DIS
LIN {X -0.196,Y -426.355,Z 358.472,A 0.000,B 0.000,C 90.000,E1 84.951} C_DIS
LIN {X 0.015,Y -407.959,Z 358.454,A 0.000,B 0.000,C 90.000,E1 81.659} C_DIS
LIN {X -0.124,Y -396.267,Z 358.441,A 0.000,B 0.000,C 90.000,E1 79.454} C_DIS
LIN {X -0.060,Y -386.062,Z 358.430,A 0.000,B 0.000,C 90.000,E1 77.465} C_DIS
LIN {X -0.114,Y -374.442,Z 358.418,A 0.000,B 0.000,C 90.000,E1 75.172} C_DIS
LIN {X -0.183,Y -361.408,Z 358.403,A 0.000,B 0.000,C 90.000,E1 72.543} C_DIS
LIN {X -0.011,Y -351.271,Z 358.391,A 0.000,B 0.000,C 90.000,E1 70.423} C_DIS
LIN {X 0.079,Y -337.156,Z 358.374,A 0.000,B 0.000,C 90.000,E1 67.358} C_DIS
LIN {X -0.132,Y -325.320,Z 358.359,A 0.000,B 0.000,C 90.000,E1 64.588} C_DIS
LIN {X 0.058,Y -314.495,Z 358.343,A 0.000,B 0.000,C 90.000,E1 61.691} C_DIS
LIN {X 0.043,Y -302.064,Z 358.323,A 0.000,B 0.000,C 90.000,E1 58.122} C_DIS
LIN {X 0.023,Y -291.625,Z 358.305,A 0.000,B 0.000,C 90.000,E1 54.815} C_DIS
LIN {X -0.039,Y -282.078,Z 358.286,A 0.000,B 0.000,C 90.000,E1 51.457} C_DIS
LIN {X 0.087,Y -274.567,Z 358.271,A 0.000,B 0.000,C 90.000,E1 48.690} C_DIS
LIN {X 0.033,Y -268.865,Z 358.259,A 0.000,B 0.000,C 90.000,E1 46.620} C_DIS
LIN {X 0.152,Y -261.293,Z 358.243,A 0.000,B 0.000,C 90.000,E1 43.785} C_DIS
LIN {X -0.088,Y -253.707,Z 358.228,A 0.000,B 0.000,C 90.000,E1 40.987} C_DIS
LIN {X -0.127,Y -247.834,Z 358.216,A 0.000,B 0.000,C 90.000,E1 38.830} C_DIS
LIN {X -0.049,Y -239.957,Z 358.199,A 0.000,B 0.000,C 90.000,E1 35.884} C_DIS
LIN {X 0.074,Y -232.310,Z 358.183,A 0.000,B 0.000,C 90.000,E1 32.880} C_DIS
LIN {X -0.050,Y -223.165,Z 358.162,A 0.000,B 0.000,C 90.000,E1 29.127} C_DIS
LIN {X -0.092,Y -215.022,Z 358.140,A 0.000,B 0.000,C 90.000,E1 25.283} C_DIS
LIN {X -0.091,Y -209.156,Z 358.123,A 0.000,B 0.000,C 90.000,E1 22.153} C_DIS
LIN {X -0.012,Y -204.034,Z 358.105,A 0.000,B 0.000,C 90.000,E1 18.960} C_DIS
LIN {X -0.030,Y -198.504,Z 358.083,A 0.000,B 0.000,C 90.000,E1 14.954} C_DIS
LIN {X -0.029,Y -194.017,Z 358.060,A 0.000,B 0.000,C 90.000,E1 10.894} C_DIS
LIN {X 0.036,Y -190.662,Z 358.038,A 0.000,B 0.000,C 90.000,E1 6.777} C_DIS
LIN {X -0.086,Y -188.054,Z 358.006,A 0.000,B 0.000,C 90.000,E1 1.031} C_DIS
LIN {X 0.028,Y -189.261,Z 357.942,A 0.000,B 0.000,C 90.000,E1 349.567} C_DIS
LIN {X -0.031,Y -192.131,Z 357.915,A 0.000,B 0.000,C 90.000,E1 344.629} C_DIS
LIN {X 0.071,Y -195.723,Z 357.892,A 0.000,B 0.000,C 90.000,E1 340.496} C_DIS
LIN {X 0.059,Y -200.447,Z 357.869,A 0.000,B 0.000,C 90.000,E1 336.433} C_DIS
LIN {X 0.058,Y -206.202,Z 357.847,A 0.000,B 0.000,C 90.000,E1 332.410} C_DIS
LIN {X -0.008,Y -212.930,Z 357.825,A 0.000,B 0.000,C 90.000,E1 328.456} C_DIS
LIN {X -0.084,Y -220.301,Z 357.803,A 0.000,B 0.000,C 90.000,E1 324.562} C_DIS
LIN {X 0.042,Y -228.552,Z 357.782,A 0.000,B 0.000,C 90.000,E1 320.678} C_DIS
LIN {X 0.090,Y -235.944,Z 357.765,A 0.000,B 0.000,C 90.000,E1 317.634} C_DIS
LIN {X 0.139,Y -245.299,Z 357.746,A 0.000,B 0.000,C 90.000,E1 314.271} C_DIS
LIN {X 0.139,Y -255.929,Z 357.728,A 0.000,B 0.000,C 90.000,E1 310.987} C_DIS
LIN {X -0.033,Y -267.334,Z 357.710,A 0.000,B 0.000,C 90.000,E1 307.810} C_DIS
LIN {X -0.005,Y -279.765,Z 357.693,A 0.000,B 0.000,C 90.000,E1 304.659} C_DIS
LIN {X -0.017,Y -293.527,Z 357.676,A 0.000,B 0.000,C 90.000,E1 301.592} C_DIS
LIN {X -0.053,Y -310.684,Z 357.657,A 0.000,B 0.000,C 90.000,E1 298.281} C_DIS
LIN {X -0.094,Y -320.216,Z 357.648,A 0.000,B 0.000,C 90.000,E1 296.668} C_DIS
LIN {X -0.131,Y -341.255,Z 357.631,A 0.000,B 0.000,C 90.000,E1 293.515} C_DIS
LIN {X -0.031,Y -356.922,Z 357.619,A 0.000,B 0.000,C 90.000,E1 291.354} C_DIS
LIN {X -0.039,Y -373.337,Z 357.607,A 0.000,B 0.000,C 90.000,E1 289.268} C_DIS
LIN {X 0.032,Y -396.091,Z 357.593,A 0.000,B 0.000,C 90.000,E1 286.677} C_DIS
LIN {X 0.088,Y -413.886,Z 357.582,A 0.000,B 0.000,C 90.000,E1 284.773} C_DIS
LIN {X -0.004,Y -426.495,Z 357.575,A 0.000,B 0.000,C 90.000,E1 283.467} C_DIS
LIN {X 0.165,Y -433.852,Z 357.570,A 0.000,B 0.000,C 90.000,E1 282.647} C_DIS
LIN {X -0.112,Y -440.783,Z 357.566,A 0.000,B 0.000,C 90.000,E1 281.883} C_DIS
LIN {X 0.008,Y -447.263,Z 357.562,A 0.000,B 0.000,C 90.000,E1 281.074} C_DIS
LIN {X 0.090,Y -455.120,Z 357.556,A 0.000,B 0.000,C 90.000,E1 280.018} C_DIS
LIN {X 0.183,Y -462.414,Z 357.550,A 0.000,B 0.000,C 90.000,E1 278.973} C_DIS
LIN {X -0.167,Y -469.003,Z 357.544,A 0.000,B 0.000,C 90.000,E1 277.992} C_DIS
LIN {X 0.086,Y -475.169,Z 357.539,A 0.000,B 0.000,C 90.000,E1 276.947} C_DIS
LIN {X -0.124,Y -480.605,Z 357.533,A 0.000,B 0.000,C 90.000,E1 275.967} C_DIS
LIN {X -0.013,Y -482.958,Z 357.530,A 0.000,B 0.000,C 90.000,E1 275.454} C_DIS
LIN {X 0.162,Y -484.986,Z 357.528,A 0.000,B 0.000,C 90.000,E1 274.935} C_DIS
LIN {X -0.142,Y -486.621,Z 357.525,A 0.000,B 0.000,C 90.000,E1 274.473} C_DIS
LIN {X 0.047,Y -487.839,Z 357.522,A 0.000,B 0.000,C 90.000,E1 273.955} C_DIS
LIN {X 0.214,Y -488.675,Z 357.519,A 0.000,B 0.000,C 90.000,E1 273.440} C_DIS
LIN {X -0.071,Y -489.163,Z 357.517,A 0.000,B 0.000,C 90.000,E1 272.980} C_DIS
LIN {X 0.113,Y -489.370,Z 357.514,A 0.000,B 0.000,C 90.000,E1 272.465} C_DIS
LIN {X -0.188,Y -489.292,Z 357.511,A 0.000,B 0.000,C 90.000,E1 272.007} C_DIS
LIN {X 0.017,Y -488.934,Z 357.508,A 0.000,B 0.000,C 90.000,E1 271.489} C_DIS
LIN {X 0.207,Y -488.269,Z 357.506,A 0.000,B 0.000,C 90.000,E1 270.974} C_DIS
LIN {X -0.093,Y -487.264,Z 357.503,A 0.000,B 0.000,C 90.000,E1 270.516} C_DIS
LIN {X 0.092,Y -485.834,Z 357.500,A 0.000,B 0.000,C 90.000,E1 270.000} C_DIS
LIN {X 0.112,Y -482.840,Z 357.496,A 0.000,B 0.000,C 90.000,E1 269.255} C_DIS
LIN {X -0.209,Y -479.982,Z 357.493,A 0.000,B 0.000,C 90.000,E1 268.797} C_DIS
LIN {X 0.105,Y -478.321,Z 357.492,A 0.000,B 0.000,C 90.000,E1 268.511} C_DIS
LIN {X -0.223,Y -474.124,Z 357.489,A 0.000,B 0.000,C 90.000,E1 268.051} C_DIS
LIN {X 0.069,Y -471.639,Z 357.488,A 0.000,B 0.000,C 90.000,E1 267.764} C_DIS
LIN {X -0.083,Y -465.890,Z 357.485,A 0.000,B 0.000,C 90.000,E1 267.306} C_DIS
LIN {X -0.055,Y -462.647,Z 357.484,A 0.000,B 0.000,C 90.000,E1 267.078} C_DIS
LIN {X -0.234,Y -459.404,Z 357.483,A 0.000,B 0.000,C 90.000,E1 266.906} C_DIS
